(* CoDeSys 2.3.9.62 project: furrestaurantecasidefinitivo.pro *)
(* Libraries: Standard.lib 4.10.05 13:14:46, IecSfc.lib 2.6.14 11:37:46, SYSLIBCALLBACK.LIB 26.9.08 17:43:52 *)

(* Global variable list: Global_Variables *)
VAR_GLOBAL
	(*VISUALIZACION_PLATOS*)
	plato:ARRAY [1..8] OF elemento2d;
	pistonx:INT;
	vpist:INT := 3;
	velp:INT := 3;
		(*ACTUADORES CINTAS*)
		CIN_ENT_COC:BOOL;
		CIN_CLA:BOOL;
		CIN_H1:BOOL;
		CIN_H2:BOOL;
		CIN_H3:BOOL;
		CIN_SERVIR:BOOL;
		CIN_H1_A_REAL:BOOL;
		CIN_H2_A_REAL:BOOL;
		CIN_H3_A_REAL:BOOL;
		CIN_REALIM:BOOL;
		CIN_COLA_SERV:BOOL;
		(*ACTUADORES PISTON Y PROCESOS*)
		PISCLA_MAS:BOOL;
		PISCLA_MENOS:BOOL;
		AGARRAR:BOOL;
		H1:BOOL;
		H2:BOOL;
		H3:BOOL;
		DISP_PLATO:BOOL;
			(*BOTONERA CONTROL PLATOS*)
			b1:BOOL;
			b2:BOOL;
			b3:BOOL;
			b4:BOOL;
			b5:BOOL;
			b6:BOOL;
			b7:BOOL;
			b8:BOOL;
			br1:BOOL;
			br2:BOOL;
			br3:BOOL;
			blisto:BOOL;
			bup:BOOL;
			bdown:BOOL;
			bleft:BOOL;
			bright:BOOL;
			bhide:BOOL;
			vel: INT :=1 ;
		(*SENSORES CINTAS*)
		ENT_COC:BOOL;
		SEM_ENT_COC:BOOL;
		SEM_SAL_REAL:BOOL;
		S_CLA:ARRAY [1..8] OF BOOL;
		ENT_CLA:BOOL;
		ENT_H1:BOOL;
		ENT_H2:BOOL;
		ENT_H3:BOOL;
		ENT_SERVIR:BOOL;
		ESPERA_H1:BOOL;
		ESPERA_H2:BOOL;
		ESPERA_H3:BOOL;
		ENT_REAL1:BOOL;
		ENT_REAL2:BOOL;
		ENT_REAL3:BOOL;
		SEM_H2_R:BOOL;
		SEM_H2_V:BOOL;
		SEM_H2:BOOL;
		SEM_H1_R:BOOL;
		SEM_H1_V:BOOL;
		SEM_H1:BOOL;
		SAL_R:BOOL;
		ENT_TER:BOOL;
		TER_1:BOOL;
		TER_2:BOOL;
		TER_3:BOOL;
		(*SENSORES PISTON Y PROCESOS*)
		S_H1:BOOL;
		S_H2:BOOL;
		S_H3:BOOL;
		FC_PISCLA:BOOL;
		(*INFOPLATO*)

	(*VISUALIZACIÓN AGVs*)
	x1:INT:=130;
	y1:INT;
	x2:INT:=330;
	y2:INT;

		(*ACTUADORES AGVS*)
		SERVIR_PLATO1:BOOL;
		SERVIR_PLATO2:BOOL;
		CARGAR_PLATO:ARRAY [1..3] OF BOOL;

		(*SENSORES AGVs*)
		CARGADO1:BOOL;
		CARGADO2:BOOL;

		(*ACTUADORES SALÓN*)
		MARCHA1:BOOL;
		MARCHA2:BOOL;
		BIF_ARRIBA1:BOOL;
		BIF_ABAJO1:BOOL;
		BIF_ARRIBA2:BOOL;
		BIF_ABAJO2:BOOL;
		SEM_M1:BOOL;
		SEM_M2:BOOL;
		SEM_M3:BOOL;
		SEM_M4:BOOL;
		SEM_M5:BOOL;
		SEM_M6:BOOL;
		SEM_M7:BOOL;
		SEM_M8:BOOL;

		(*SENSORES SALÓN*)

		PC1_1:BOOL;
		PC1_2:BOOL;
		PR1_3:BOOL;
		PR1_2:BOOL;
		PR1_1:BOOL;
		BIF1_12:BOOL;
		BIF1_34:BOOL;
		BIF1_56:BOOL;
		BIF1_78:BOOL;

		PC2_1:BOOL;
		PC2_2:BOOL;
		PR2_3:BOOL;
		PR2_2:BOOL;
		PR2_1:BOOL;
		BIF2_12:BOOL;
		BIF2_34:BOOL;
		BIF2_56:BOOL;
		BIF2_78:BOOL;

		PS_1:BOOL;
		PS_2:BOOL;
		PS_3:BOOL;
		PS_4:BOOL;
		PS_5:BOOL;
		PS_6:BOOL;
		PS_7:BOOL;
		PS_8:BOOL;

		SS_PS_1:BOOL;
		SS_PS_2:BOOL;
		SS_PS_3:BOOL;
		SS_PS_4:BOOL;
		SS_PS_5:BOOL;
		SS_PS_6:BOOL;
		SS_PS_7:BOOL;
		SS_PS_8:BOOL;
		SS_F:BOOL;

	(*VISUALIZACION SALON*)
	ESTADO_MESA:ARRAY [1..8] OF BOOL;

		(*COLAS*)
		PENDIENTES_ENTRAR:ARRAY [1..20] OF INT;
		MESA_PEDIDO:ARRAY [1..20,1..2] OF INT;
		PEDIDO1:BOOL;
		PEDIDO2:BOOL;
		PEDIDO3:BOOL;
		MESA1:BOOL;
		MESA2:BOOL;
		MESA3:BOOL;
		MESA4:BOOL;
		MESA5:BOOL;
		MESA6:BOOL;
		MESA7:BOOL;
		MESA8:BOOL;

		(*BOTONERA COLAS*)
		B_CANCELAR:BOOL;
		B_PEDIR:BOOL;
		B_MESA:ARRAY [1..8] OF BOOL;
		B_PEDIDO:ARRAY [1..3] OF BOOL;




(*VARIABLES AUXILIARES*)
	LLENO:BOOL;
	ESPERA_ENTCOC:BOOL;
	ESPERA_CLA:BOOL;
	ESPERA_CINH1:BOOL;
	ESPERA_CINH2:BOOL;
	ESPERA_CINH3:BOOL;
	ESPERA_REAL:BOOL;
	ESPERA_SERVIR:BOOL;
	PASAH1:BOOL;
	PASAH2:BOOL;
	PASAH3:BOOL;
	H1OK:BOOL;
	H2OK:BOOL;
	H3OK:BOOL;
	SALE_REAL:BOOL;
	DIR_PISTON:ARRAY[1..8] OF INT;
	TDISP:BOOL;
	PLATO_SEM_H2:BOOL;
	PLATO_SEM_H1:BOOL;
	OC2:BOOL;
	OC1:BOOL;
	SCLAAUX:BOOL;
	REALIMENTANDO:BOOL;
	TIEMPODISP:BOOL;
END_VAR

(* Data type *)
TYPE elemento2d :
STRUCT
	x:INT;
	y:INT;
	P1:INT;
	P2:INT;
	P3:INT;
	REC:INT;
	on:BOOL;
	listo:BOOL;
	receta:STRING(5); (*temporal, solo se usara en la visualizacion*)
END_STRUCT
END_TYPE

(* POU PLC_PRG, ST *)
PROGRAM PLC_PRG
VAR
END_VAR
INFO_PLATOS;
CONTADORES;
SEMAFORO_SALIDA_H2;
SEMAFORO_SALIDA_H1;
SEMAFORO_ENTCOC;
PROCESOS;
PISTON;
CONTROL_CINTAS;
CINTA_COLA;
VIS_BOTON_PLATO;
VIS_MESAS;
VIS_PISTON;
VIS_CINTAS_PLATO;
VIS_AGV;
COLAS_PEDIDOS;
END_PROGRAM

(* POU INFO_PLATOS, ST *)
PROGRAM INFO_PLATOS
VAR
	R1:ARRAY[1..3] OF INT:=1,2,3;
	R2:ARRAY[1..3] OF INT:=2,1,3;
	R3:ARRAY[1..3] OF INT:=3,2,1;
	FS_SCLA:ARRAY[1..8] OF BOOL;
	i:INT:=1;
	i2:INT:=1;
	j:INT:=1;
	k:INT:=1;
	t:INT:=1;
	p:INT:=1;
	FLAG_DIR:BOOL;
	DISPLIBRE: BOOL:=TRUE;
	FS_DISPPLATO: BOOL;
	FB_AGARRAR:BOOL;
END_VAR
(*Asignación de receta a plato desde cola y actualización de la misma*)

IF FS_DISPPLATO=TRUE THEN
	FS_DISPPLATO:=FALSE;
	DISP_PLATO:=FALSE;
END_IF

IF NOT DISPLIBRE AND TIEMPODISP THEN
	DISPLIBRE:=TRUE;
END_IF

IF PENDIENTES_ENTRAR[1]<>0 THEN
	plato[j].REC:=PENDIENTES_ENTRAR[1];
	FOR i:=2 TO 20 BY 1 DO
		PENDIENTES_ENTRAR[i-1]:=PENDIENTES_ENTRAR[i];
	END_FOR
	PENDIENTES_ENTRAR[20]:=0;

	IF plato[j].REC=1 THEN
		plato[j].P1:=R1[1];
		plato[j].P2:=R1[2];
		plato[j].P3:=R1[3];
		plato[j].receta:='R1';
	ELSIF plato[j].REC=2 THEN
		plato[j].P1:=R2[1];
		plato[j].P2:=R2[2];
		plato[j].P3:=R2[3];
		plato[j].receta:='R2';
	ELSIF plato[j].REC=3 THEN
		plato[j].P1:=R3[1];
		plato[j].P2:=R3[2];
		plato[j].P3:=R3[3];
		plato[j].receta:='R3';
	END_IF
	IF j<8 THEN
		j:=j+1;
	ELSE
		j:=1;
	END_IF
END_IF

IF NOT LLENO AND FC_PISCLA AND NOT ENT_CLA AND DISPLIBRE AND plato[i2].P1<>0 THEN
	DISP_PLATO:=TRUE;
	FS_DISPPLATO:=TRUE;
	DISPLIBRE:=FALSE;
	IF i2<8 THEN
		i2:=i2+1;
	ELSE
		i2:=1;
	END_IF
END_IF



(*Manejo del sensor de clasificación S_CLA y comunicación con el pistón*)

FOR t:=1 TO 8 BY 1 DO
	IF S_CLA[t]=TRUE AND FS_SCLA[t]=FALSE THEN
		FS_SCLA[t]:=TRUE;
		IF plato[t].P1<>0 THEN
			FOR k:=1 TO 8 BY 1 DO
				IF DIR_PISTON[k]=0 AND FLAG_DIR=FALSE THEN
					DIR_PISTON[k]:=plato[t].P1;
					FLAG_DIR:=TRUE;
				END_IF
			END_FOR
			FLAG_DIR:=FALSE;
			plato[t].P1:=0;
		ELSIF plato[t].P1=0 AND plato[t].P2<>0 THEN
			FOR k:=1 TO 8 BY 1 DO
				IF DIR_PISTON[k]=0 AND FLAG_DIR=FALSE THEN
					DIR_PISTON[k]:=plato[t].P2;
					FLAG_DIR:=TRUE;
				END_IF
			END_FOR
			FLAG_DIR:=FALSE;
			plato[t].P2:=0;
		ELSIF plato[t].P1=0 AND plato[t].P2=0 AND plato[t].P3<>0 THEN
			FOR k:=1 TO 8 BY 1 DO
				IF DIR_PISTON[k]=0 AND FLAG_DIR=FALSE THEN
					DIR_PISTON[k]:=plato[t].P3;
					FLAG_DIR:=TRUE;
				END_IF
			END_FOR
			FLAG_DIR:=FALSE;
			plato[t].P3:=0;
		ELSIF plato[t].P1=0 AND plato[t].P2=0 AND plato[t].P3=0 AND plato[t].REC<>0 THEN
			FOR k:=1 TO 8 BY 1 DO
				IF DIR_PISTON[k]=0 AND FLAG_DIR=FALSE THEN
					DIR_PISTON[k]:=4;
					FLAG_DIR:=TRUE;
					plato[t].listo:=TRUE;
				END_IF
			END_FOR
			FLAG_DIR:=FALSE;
			plato[t].REC:=0;
		END_IF
	ELSIF S_CLA[t]=FALSE THEN
		FS_SCLA[t]:=FALSE;
	END_IF
END_FOR

(*Manejo de la cola del pistón*)




IF NOT AGARRAR AND NOT FB_AGARRAR THEN
	FOR p:=2 TO 8 BY 1 DO
		DIR_PISTON[p-1]:=DIR_PISTON[p];
	END_FOR
	DIR_PISTON[8]:=0;
	FB_AGARRAR:=TRUE;
ELSIF AGARRAR THEN
	FB_AGARRAR:=FALSE;
END_IF
END_PROGRAM

(* POU CONTADORES, LD *)
PROGRAM CONTADORES
VAR
	NUM_ENTCOC: CTUD;
	NUM_COCINA: CTUD;
	NUM_CLA: CTUD;
	FB_ENTCOC1: F_TRIG;
	FB_ENTCOC2: F_TRIG;
	NUM_H1: CTUD;
	NUM_H2: CTUD;
	NUM_H3: CTUD;
	NUM_REAL: CTUD;
	RET_SALREAL: TOF;
	FS_ENTH3: R_TRIG;
	FS_ENTH2: R_TRIG;
	FS_ENTH1: R_TRIG;
	FS_SALEREAL: R_TRIG;
	FS_ENTSERVIR: R_TRIG;
	NUM_SERVIR: CTUD;
	SEPARACION_PLATOS_DISP: TOF;
	ENTRA_SMF_H2: R_TRIG;
	NUM_SMF_H2: CTUD;
	ENTRA_SMF_H1: R_TRIG;
	NUM_SMF_H1: CTUD;
	TSEMAFORO2: TON;
	TSEMAFORO1: TON;
	FS_ENTREAL1: R_TRIG;
	FS_ENTREAL2: R_TRIG;
	FS_ENTREAL3: R_TRIG;
	FB_SALR: F_TRIG;
	FB_DISPPLATO: F_TRIG;
	tiempo_disp: TON;
END_VAR
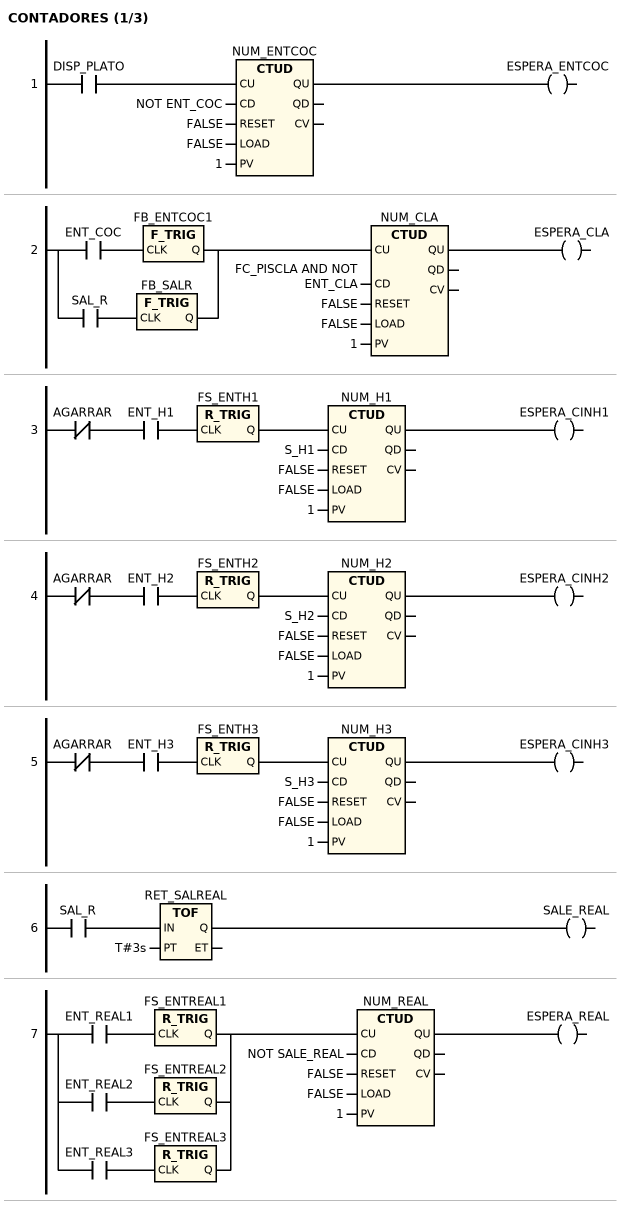
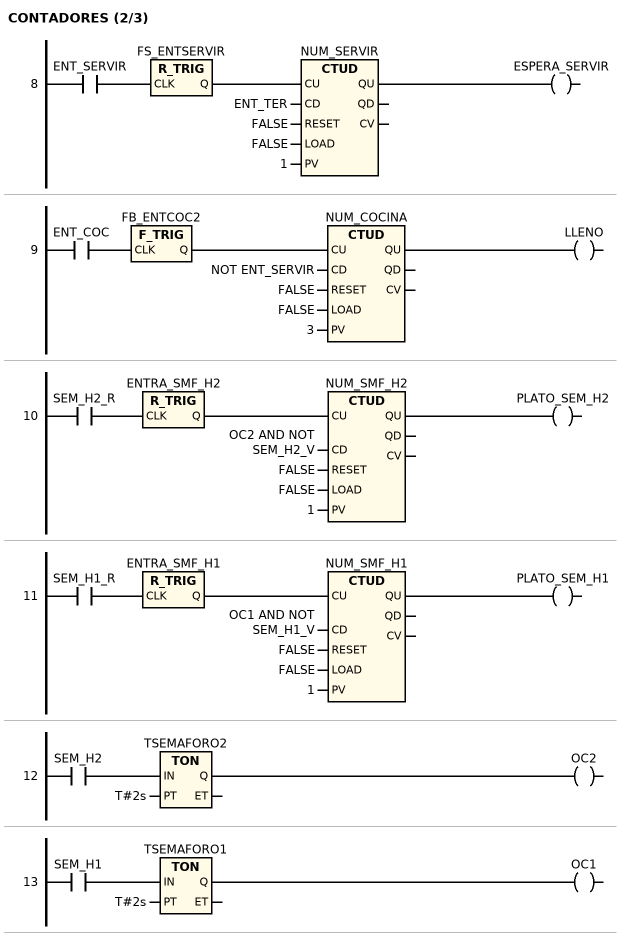
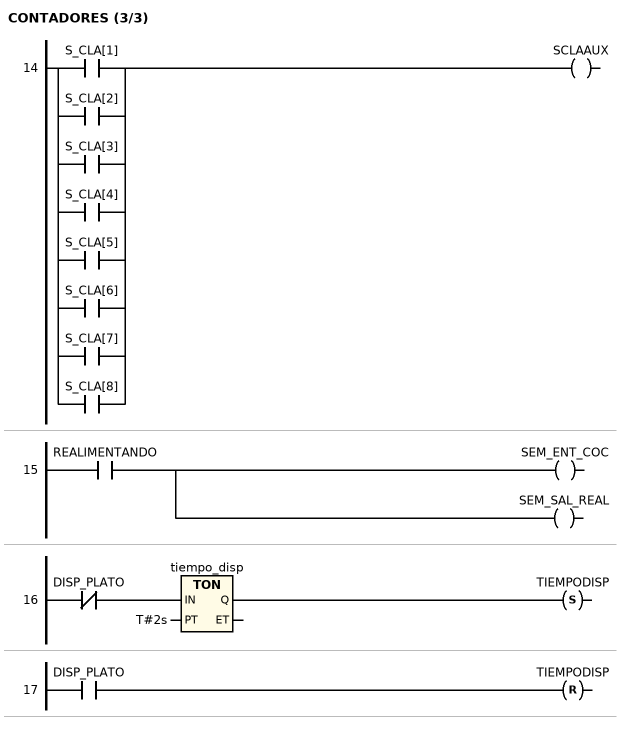
_LD_ (* Ladder Diagram *)
NETWORK 1
	[DISP_PLATO] - NUM_ENTCOC:CTUD(CU: *, CD: NOT ENT_COC, RESET: FALSE, LOAD: FALSE, PV: 1) --- (ESPERA_ENTCOC)
NETWORK 2
	{ [ENT_COC] - FB_ENTCOC1:F_TRIG(CLK: *) | [SAL_R] - FB_SALR:F_TRIG(CLK: *) } - NUM_CLA:CTUD(CU: *, CD: FC_PISCLA AND NOT ENT_CLA, RESET: FALSE, LOAD: FALSE, PV: 1) --- (ESPERA_CLA)
NETWORK 3
	[/AGARRAR] - [ENT_H1] - FS_ENTH1:R_TRIG(CLK: *) - NUM_H1:CTUD(CU: *, CD: S_H1, RESET: FALSE, LOAD: FALSE, PV: 1) --- (ESPERA_CINH1)
NETWORK 4
	[/AGARRAR] - [ENT_H2] - FS_ENTH2:R_TRIG(CLK: *) - NUM_H2:CTUD(CU: *, CD: S_H2, RESET: FALSE, LOAD: FALSE, PV: 1) --- (ESPERA_CINH2)
NETWORK 5
	[/AGARRAR] - [ENT_H3] - FS_ENTH3:R_TRIG(CLK: *) - NUM_H3:CTUD(CU: *, CD: S_H3, RESET: FALSE, LOAD: FALSE, PV: 1) --- (ESPERA_CINH3)
NETWORK 6
	[SAL_R] - RET_SALREAL:TOF(IN: *, PT: T#3s) --- (SALE_REAL)
NETWORK 7
	{ [ENT_REAL1] - FS_ENTREAL1:R_TRIG(CLK: *) | [ENT_REAL2] - FS_ENTREAL2:R_TRIG(CLK: *) | [ENT_REAL3] - FS_ENTREAL3:R_TRIG(CLK: *) } - NUM_REAL:CTUD(CU: *, CD: NOT SALE_REAL, RESET: FALSE, LOAD: FALSE, PV: 1) --- (ESPERA_REAL)
NETWORK 8
	[ENT_SERVIR] - FS_ENTSERVIR:R_TRIG(CLK: *) - NUM_SERVIR:CTUD(CU: *, CD: ENT_TER, RESET: FALSE, LOAD: FALSE, PV: 1) --- (ESPERA_SERVIR)
NETWORK 9
	[ENT_COC] - FB_ENTCOC2:F_TRIG(CLK: *) - NUM_COCINA:CTUD(CU: *, CD: NOT ENT_SERVIR, RESET: FALSE, LOAD: FALSE, PV: 3) --- (LLENO)
NETWORK 10
	[SEM_H2_R] - ENTRA_SMF_H2:R_TRIG(CLK: *) - NUM_SMF_H2:CTUD(CU: *, CD: OC2 AND NOT SEM_H2_V, RESET: FALSE, LOAD: FALSE, PV: 1) --- (PLATO_SEM_H2)
NETWORK 11
	[SEM_H1_R] - ENTRA_SMF_H1:R_TRIG(CLK: *) - NUM_SMF_H1:CTUD(CU: *, CD: OC1 AND NOT SEM_H1_V, RESET: FALSE, LOAD: FALSE, PV: 1) --- (PLATO_SEM_H1)
NETWORK 12
	[SEM_H2] - TSEMAFORO2:TON(IN: *, PT: T#2s) --- (OC2)
NETWORK 13
	[SEM_H1] - TSEMAFORO1:TON(IN: *, PT: T#2s) --- (OC1)
NETWORK 14
	{ [S_CLA[1]] | [S_CLA[2]] | [S_CLA[3]] | [S_CLA[4]] | [S_CLA[5]] | [S_CLA[6]] | [S_CLA[7]] | [S_CLA[8]] } --- (SCLAAUX)
NETWORK 15
	[REALIMENTANDO] --- (SEM_ENT_COC) (SEM_SAL_REAL)
NETWORK 16
	[/DISP_PLATO] - tiempo_disp:TON(IN: *, PT: T#2s) --- (S TIEMPODISP)
NETWORK 17
	[DISP_PLATO] --- (R TIEMPODISP)
_END_LD_
(* the same logic as Structured Text *)
(* Network 1 *)
NUM_ENTCOC(CU := DISP_PLATO, CD := NOT ENT_COC, RESET := FALSE, LOAD := FALSE, PV := 1);
ESPERA_ENTCOC := NUM_ENTCOC.QU;
(* Network 2 *)
FB_ENTCOC1(CLK := ENT_COC);
FB_SALR(CLK := SAL_R);
NUM_CLA(CU := FB_ENTCOC1.Q OR FB_SALR.Q, CD := FC_PISCLA AND NOT ENT_CLA, RESET := FALSE, LOAD := FALSE, PV := 1);
ESPERA_CLA := NUM_CLA.QU;
(* Network 3 *)
FS_ENTH1(CLK := NOT AGARRAR AND ENT_H1);
NUM_H1(CU := FS_ENTH1.Q, CD := S_H1, RESET := FALSE, LOAD := FALSE, PV := 1);
ESPERA_CINH1 := NUM_H1.QU;
(* Network 4 *)
FS_ENTH2(CLK := NOT AGARRAR AND ENT_H2);
NUM_H2(CU := FS_ENTH2.Q, CD := S_H2, RESET := FALSE, LOAD := FALSE, PV := 1);
ESPERA_CINH2 := NUM_H2.QU;
(* Network 5 *)
FS_ENTH3(CLK := NOT AGARRAR AND ENT_H3);
NUM_H3(CU := FS_ENTH3.Q, CD := S_H3, RESET := FALSE, LOAD := FALSE, PV := 1);
ESPERA_CINH3 := NUM_H3.QU;
(* Network 6 *)
RET_SALREAL(IN := SAL_R, PT := T#3s);
SALE_REAL := RET_SALREAL.Q;
(* Network 7 *)
FS_ENTREAL1(CLK := ENT_REAL1);
FS_ENTREAL2(CLK := ENT_REAL2);
FS_ENTREAL3(CLK := ENT_REAL3);
NUM_REAL(CU := FS_ENTREAL1.Q OR FS_ENTREAL2.Q OR FS_ENTREAL3.Q, CD := NOT SALE_REAL, RESET := FALSE, LOAD := FALSE, PV := 1);
ESPERA_REAL := NUM_REAL.QU;
(* Network 8 *)
FS_ENTSERVIR(CLK := ENT_SERVIR);
NUM_SERVIR(CU := FS_ENTSERVIR.Q, CD := ENT_TER, RESET := FALSE, LOAD := FALSE, PV := 1);
ESPERA_SERVIR := NUM_SERVIR.QU;
(* Network 9 *)
FB_ENTCOC2(CLK := ENT_COC);
NUM_COCINA(CU := FB_ENTCOC2.Q, CD := NOT ENT_SERVIR, RESET := FALSE, LOAD := FALSE, PV := 3);
LLENO := NUM_COCINA.QU;
(* Network 10 *)
ENTRA_SMF_H2(CLK := SEM_H2_R);
NUM_SMF_H2(CU := ENTRA_SMF_H2.Q, CD := OC2 AND NOT SEM_H2_V, RESET := FALSE, LOAD := FALSE, PV := 1);
PLATO_SEM_H2 := NUM_SMF_H2.QU;
(* Network 11 *)
ENTRA_SMF_H1(CLK := SEM_H1_R);
NUM_SMF_H1(CU := ENTRA_SMF_H1.Q, CD := OC1 AND NOT SEM_H1_V, RESET := FALSE, LOAD := FALSE, PV := 1);
PLATO_SEM_H1 := NUM_SMF_H1.QU;
(* Network 12 *)
TSEMAFORO2(IN := SEM_H2, PT := T#2s);
OC2 := TSEMAFORO2.Q;
(* Network 13 *)
TSEMAFORO1(IN := SEM_H1, PT := T#2s);
OC1 := TSEMAFORO1.Q;
(* Network 14 *)
SCLAAUX := S_CLA[1] OR S_CLA[2] OR S_CLA[3] OR S_CLA[4] OR S_CLA[5] OR S_CLA[6] OR S_CLA[7] OR S_CLA[8];
(* Network 15 *)
SEM_ENT_COC := REALIMENTANDO;
SEM_SAL_REAL := REALIMENTANDO;
(* Network 16 *)
tiempo_disp(IN := NOT DISP_PLATO, PT := T#2s);
IF tiempo_disp.Q THEN TIEMPODISP := TRUE; END_IF;
(* Network 17 *)
IF DISP_PLATO THEN TIEMPODISP := FALSE; END_IF;
END_PROGRAM

(* POU SEMAFORO_SALIDA_H2, SFC *)
PROGRAM SEMAFORO_SALIDA_H2
VAR
END_VAR
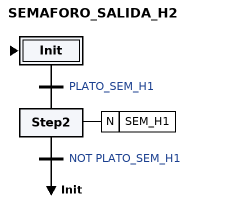
INITIAL_STEP Init:
END_STEP
TRANSITION FROM Init TO Step2 := PLATO_SEM_H1;
END_TRANSITION
STEP Step2:
	SEM_H1(N);
END_STEP
TRANSITION FROM Step2 TO Init := NOT PLATO_SEM_H1;
END_TRANSITION
END_PROGRAM

(* POU SEMAFORO_SALIDA_H1, SFC *)
PROGRAM SEMAFORO_SALIDA_H1
VAR
END_VAR
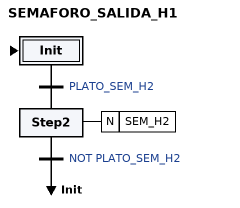
INITIAL_STEP Init:
END_STEP
TRANSITION FROM Init TO Step2 := PLATO_SEM_H2;
END_TRANSITION
STEP Step2:
	SEM_H2(N);
END_STEP
TRANSITION FROM Step2 TO Init := NOT PLATO_SEM_H2;
END_TRANSITION
END_PROGRAM

(* POU SEMAFORO_ENTCOC, SFC *)
PROGRAM SEMAFORO_ENTCOC
VAR
	FB_SALR: F_TRIG;
	FB_SCLAAUX: F_TRIG;
END_VAR
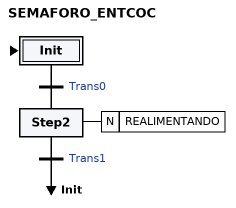
INITIAL_STEP Init:
END_STEP
TRANSITION FROM Init TO Step2 := Trans0;
END_TRANSITION
STEP Step2:
	REALIMENTANDO(N);
END_STEP
TRANSITION FROM Step2 TO Init := Trans1;
END_TRANSITION

TRANSITION Trans0:
_LD_ (* Ladder Diagram *)
NETWORK 1
	[SAL_R] - FB_SALR:F_TRIG(CLK: *)
_END_LD_
(* the same logic as Structured Text *)
(* Network 1 *)
FB_SALR(CLK := SAL_R);
Trans0 := FB_SALR.Q;
END_TRANSITION

TRANSITION Trans1:
_LD_ (* Ladder Diagram *)
NETWORK 1
	[SCLAAUX] - FB_SCLAAUX:F_TRIG(CLK: *)
_END_LD_
(* the same logic as Structured Text *)
(* Network 1 *)
FB_SCLAAUX(CLK := SCLAAUX);
Trans1 := FB_SCLAAUX.Q;
END_TRANSITION
END_PROGRAM

(* POU PROCESOS, LD *)
PROGRAM PROCESOS
VAR
	PROCESO_H1: FB_PROCESOS;
	PROCESO_H2: FB_PROCESOS;
	PROCESO_H3: FB_PROCESOS;
END_VAR
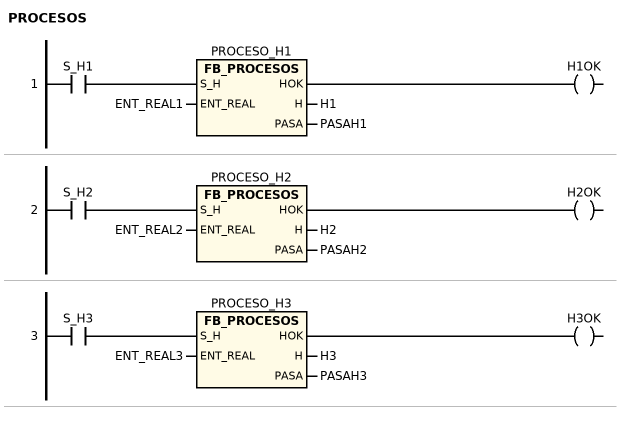
_LD_ (* Ladder Diagram *)
NETWORK 1
	[S_H1] - PROCESO_H1:FB_PROCESOS(S_H: *, ENT_REAL: ENT_REAL1, H => H1, PASA => PASAH1) --- (H1OK)
NETWORK 2
	[S_H2] - PROCESO_H2:FB_PROCESOS(S_H: *, ENT_REAL: ENT_REAL2, H => H2, PASA => PASAH2) --- (H2OK)
NETWORK 3
	[S_H3] - PROCESO_H3:FB_PROCESOS(S_H: *, ENT_REAL: ENT_REAL3, H => H3, PASA => PASAH3) --- (H3OK)
_END_LD_
(* the same logic as Structured Text *)
(* Network 1 *)
PROCESO_H1(S_H := S_H1, ENT_REAL := ENT_REAL1);
H1 := PROCESO_H1.H;
PASAH1 := PROCESO_H1.PASA;
H1OK := PROCESO_H1.HOK;
(* Network 2 *)
PROCESO_H2(S_H := S_H2, ENT_REAL := ENT_REAL2);
H2 := PROCESO_H2.H;
PASAH2 := PROCESO_H2.PASA;
H2OK := PROCESO_H2.HOK;
(* Network 3 *)
PROCESO_H3(S_H := S_H3, ENT_REAL := ENT_REAL3);
H3 := PROCESO_H3.H;
PASAH3 := PROCESO_H3.PASA;
H3OK := PROCESO_H3.HOK;
END_PROGRAM

(* POU FB_PROCESOS, SFC *)
FUNCTION_BLOCK FB_PROCESOS
VAR_INPUT
	S_H:BOOL;
	ENT_REAL:BOOL;
END_VAR
VAR_OUTPUT
	HOK:BOOL;
	H:BOOL;
	PASA:BOOL;
END_VAR
VAR
	ESPERA_PROCESO: TON;
END_VAR
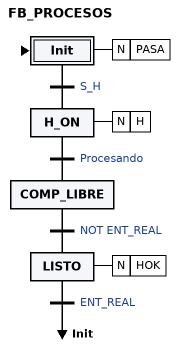
INITIAL_STEP Init:
	PASA(N);
END_STEP
TRANSITION FROM Init TO H_ON := S_H;
END_TRANSITION
STEP H_ON:
	H(N);
END_STEP
TRANSITION FROM H_ON TO COMP_LIBRE  := Procesando;
END_TRANSITION
STEP COMP_LIBRE :
END_STEP
TRANSITION FROM COMP_LIBRE  TO LISTO := NOT ENT_REAL;
END_TRANSITION
STEP LISTO:
	HOK(N);
END_STEP
TRANSITION FROM LISTO TO Init := ENT_REAL;
END_TRANSITION

TRANSITION Procesando:
_LD_ (* Ladder Diagram *)
NETWORK 1
	[H] - ESPERA_PROCESO:TON(IN: *, PT: T#5s)
_END_LD_
(* the same logic as Structured Text *)
(* Network 1 *)
ESPERA_PROCESO(IN := H, PT := T#5s);
Procesando := ESPERA_PROCESO.Q;
END_TRANSITION
END_FUNCTION_BLOCK

(* POU PISTON, SFC *)
PROGRAM PISTON
VAR
END_VAR
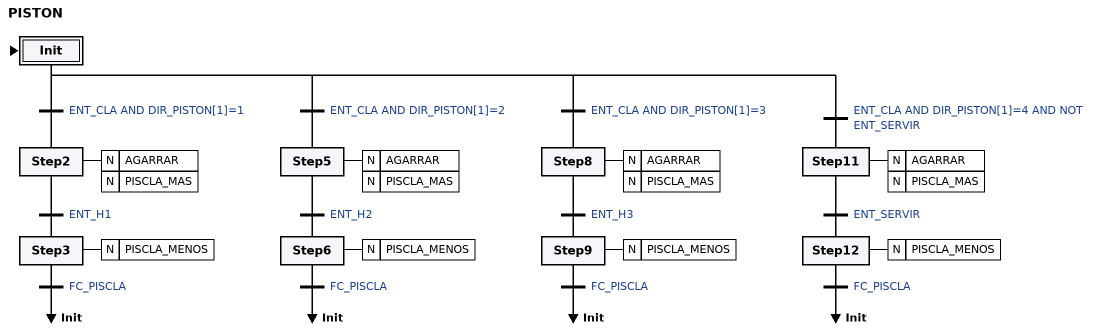
INITIAL_STEP Init:
END_STEP
TRANSITION FROM Init TO Step2 := ENT_CLA AND DIR_PISTON[1]=1;
END_TRANSITION
TRANSITION FROM Init TO Step5 := ENT_CLA AND DIR_PISTON[1]=2;
END_TRANSITION
TRANSITION FROM Init TO Step8 := ENT_CLA AND DIR_PISTON[1]=3;
END_TRANSITION
TRANSITION FROM Init TO Step11 := ENT_CLA AND DIR_PISTON[1]=4 AND NOT ENT_SERVIR;
END_TRANSITION
STEP Step2:
	AGARRAR(N);
	PISCLA_MAS(N);
END_STEP
TRANSITION FROM Step2 TO Step3 := ENT_H1;
END_TRANSITION
STEP Step3:
	PISCLA_MENOS(N);
END_STEP
TRANSITION FROM Step3 TO Init := FC_PISCLA;
END_TRANSITION
STEP Step5:
	AGARRAR(N);
	PISCLA_MAS(N);
END_STEP
TRANSITION FROM Step5 TO Step6 := ENT_H2;
END_TRANSITION
STEP Step6:
	PISCLA_MENOS(N);
END_STEP
TRANSITION FROM Step6 TO Init := FC_PISCLA;
END_TRANSITION
STEP Step8:
	AGARRAR(N);
	PISCLA_MAS(N);
END_STEP
TRANSITION FROM Step8 TO Step9 := ENT_H3;
END_TRANSITION
STEP Step9:
	PISCLA_MENOS(N);
END_STEP
TRANSITION FROM Step9 TO Init := FC_PISCLA;
END_TRANSITION
STEP Step11:
	AGARRAR(N);
	PISCLA_MAS(N);
END_STEP
TRANSITION FROM Step11 TO Step12 := ENT_SERVIR;
END_TRANSITION
STEP Step12:
	PISCLA_MENOS(N);
END_STEP
TRANSITION FROM Step12 TO Init := FC_PISCLA;
END_TRANSITION
END_PROGRAM

(* POU CONTROL_CINTAS, LD *)
PROGRAM CONTROL_CINTAS
VAR
	CINTA_H1_A_REAL: FB_CINTAS_H_A_REAL;
	CINTA_H2_A_REAL: FB_CINTAS_H_A_REAL;
	CINTA_H3_A_REAL: FB_CINTAS_H_A_REAL;
	FS_TER3: R_TRIG;
	FS_TER2: R_TRIG;
	FS_TER1: R_TRIG;
	FS_TER1_1: R_TRIG;
	FS_TER2_1: R_TRIG;
	FS_TER3_1: R_TRIG;
END_VAR
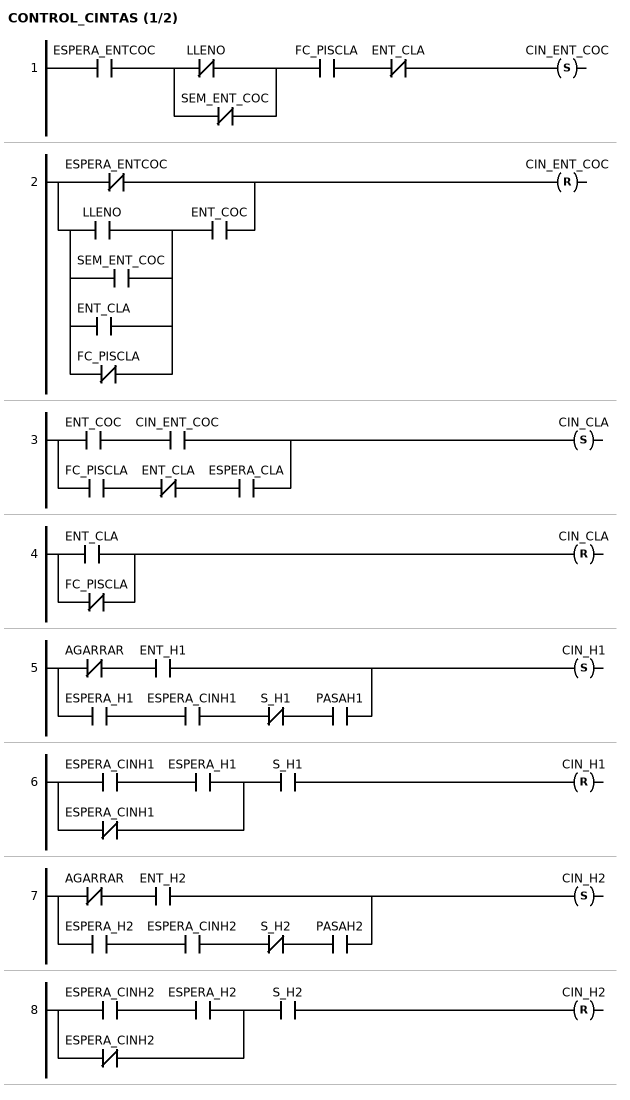
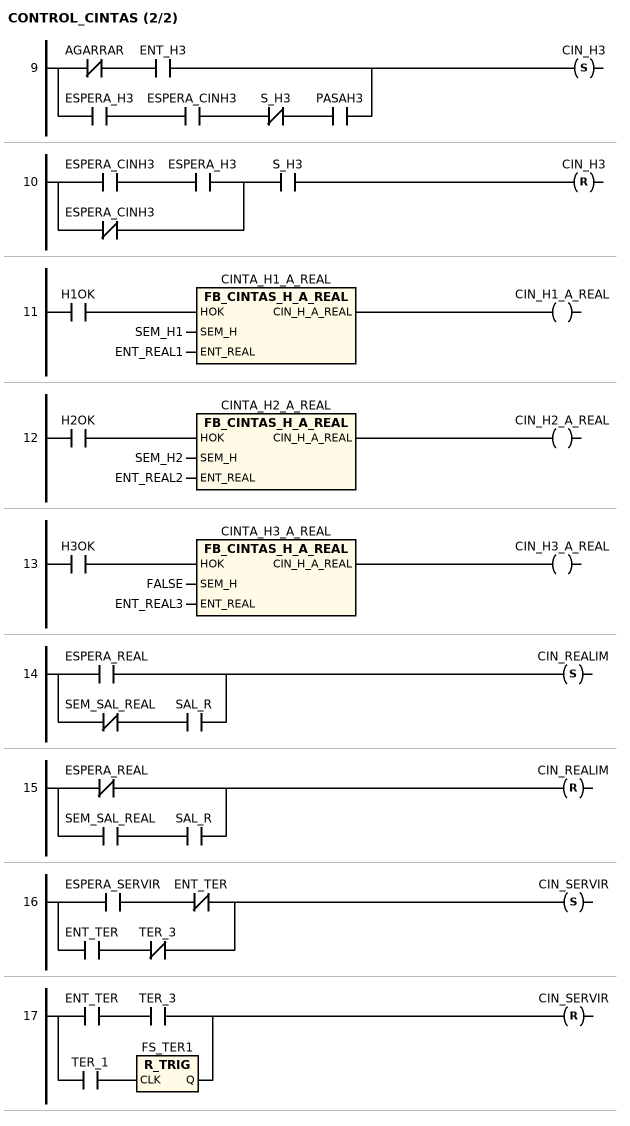
_LD_ (* Ladder Diagram *)
NETWORK 1
	[ESPERA_ENTCOC] - { [/LLENO] | [/SEM_ENT_COC] } - [FC_PISCLA] - [/ENT_CLA] --- (S CIN_ENT_COC)
NETWORK 2
	{ [/ESPERA_ENTCOC] | { [LLENO] | [SEM_ENT_COC] | [ENT_CLA] | [/FC_PISCLA] } - [ENT_COC] } --- (R CIN_ENT_COC)
NETWORK 3
	{ [ENT_COC] - [CIN_ENT_COC] | [FC_PISCLA] - [/ENT_CLA] - [ESPERA_CLA] } --- (S CIN_CLA)
NETWORK 4
	{ [ENT_CLA] | [/FC_PISCLA] } --- (R CIN_CLA)
NETWORK 5
	{ [/AGARRAR] - [ENT_H1] | [ESPERA_H1] - [ESPERA_CINH1] - [/S_H1] - [PASAH1] } --- (S CIN_H1)
NETWORK 6
	{ [ESPERA_CINH1] - [ESPERA_H1] | [/ESPERA_CINH1] } - [S_H1] --- (R CIN_H1)
NETWORK 7
	{ [/AGARRAR] - [ENT_H2] | [ESPERA_H2] - [ESPERA_CINH2] - [/S_H2] - [PASAH2] } --- (S CIN_H2)
NETWORK 8
	{ [ESPERA_CINH2] - [ESPERA_H2] | [/ESPERA_CINH2] } - [S_H2] --- (R CIN_H2)
NETWORK 9
	{ [/AGARRAR] - [ENT_H3] | [ESPERA_H3] - [ESPERA_CINH3] - [/S_H3] - [PASAH3] } --- (S CIN_H3)
NETWORK 10
	{ [ESPERA_CINH3] - [ESPERA_H3] | [/ESPERA_CINH3] } - [S_H3] --- (R CIN_H3)
NETWORK 11
	[H1OK] - CINTA_H1_A_REAL:FB_CINTAS_H_A_REAL(HOK: *, SEM_H: SEM_H1, ENT_REAL: ENT_REAL1) --- (CIN_H1_A_REAL)
NETWORK 12
	[H2OK] - CINTA_H2_A_REAL:FB_CINTAS_H_A_REAL(HOK: *, SEM_H: SEM_H2, ENT_REAL: ENT_REAL2) --- (CIN_H2_A_REAL)
NETWORK 13
	[H3OK] - CINTA_H3_A_REAL:FB_CINTAS_H_A_REAL(HOK: *, SEM_H: FALSE, ENT_REAL: ENT_REAL3) --- (CIN_H3_A_REAL)
NETWORK 14
	{ [ESPERA_REAL] | [/SEM_SAL_REAL] - [SAL_R] } --- (S CIN_REALIM)
NETWORK 15
	{ [/ESPERA_REAL] | [SEM_SAL_REAL] - [SAL_R] } --- (R CIN_REALIM)
NETWORK 16
	{ [ESPERA_SERVIR] - [/ENT_TER] | [ENT_TER] - [/TER_3] } --- (S CIN_SERVIR)
NETWORK 17
	{ [ENT_TER] - [TER_3] | [TER_1] - FS_TER1:R_TRIG(CLK: *) } --- (R CIN_SERVIR)
_END_LD_
(* the same logic as Structured Text *)
(* Network 1 *)
IF ESPERA_ENTCOC AND (NOT LLENO OR NOT SEM_ENT_COC) AND FC_PISCLA AND NOT ENT_CLA THEN CIN_ENT_COC := TRUE; END_IF;
(* Network 2 *)
IF NOT ESPERA_ENTCOC OR (LLENO OR SEM_ENT_COC OR ENT_CLA OR NOT FC_PISCLA) AND ENT_COC THEN CIN_ENT_COC := FALSE; END_IF;
(* Network 3 *)
IF ENT_COC AND CIN_ENT_COC OR FC_PISCLA AND NOT ENT_CLA AND ESPERA_CLA THEN CIN_CLA := TRUE; END_IF;
(* Network 4 *)
IF ENT_CLA OR NOT FC_PISCLA THEN CIN_CLA := FALSE; END_IF;
(* Network 5 *)
IF NOT AGARRAR AND ENT_H1 OR ESPERA_H1 AND ESPERA_CINH1 AND NOT S_H1 AND PASAH1 THEN CIN_H1 := TRUE; END_IF;
(* Network 6 *)
IF (ESPERA_CINH1 AND ESPERA_H1 OR NOT ESPERA_CINH1) AND S_H1 THEN CIN_H1 := FALSE; END_IF;
(* Network 7 *)
IF NOT AGARRAR AND ENT_H2 OR ESPERA_H2 AND ESPERA_CINH2 AND NOT S_H2 AND PASAH2 THEN CIN_H2 := TRUE; END_IF;
(* Network 8 *)
IF (ESPERA_CINH2 AND ESPERA_H2 OR NOT ESPERA_CINH2) AND S_H2 THEN CIN_H2 := FALSE; END_IF;
(* Network 9 *)
IF NOT AGARRAR AND ENT_H3 OR ESPERA_H3 AND ESPERA_CINH3 AND NOT S_H3 AND PASAH3 THEN CIN_H3 := TRUE; END_IF;
(* Network 10 *)
IF (ESPERA_CINH3 AND ESPERA_H3 OR NOT ESPERA_CINH3) AND S_H3 THEN CIN_H3 := FALSE; END_IF;
(* Network 11 *)
CINTA_H1_A_REAL(HOK := H1OK, SEM_H := SEM_H1, ENT_REAL := ENT_REAL1);
CIN_H1_A_REAL := CINTA_H1_A_REAL.CIN_H_A_REAL;
(* Network 12 *)
CINTA_H2_A_REAL(HOK := H2OK, SEM_H := SEM_H2, ENT_REAL := ENT_REAL2);
CIN_H2_A_REAL := CINTA_H2_A_REAL.CIN_H_A_REAL;
(* Network 13 *)
CINTA_H3_A_REAL(HOK := H3OK, SEM_H := FALSE, ENT_REAL := ENT_REAL3);
CIN_H3_A_REAL := CINTA_H3_A_REAL.CIN_H_A_REAL;
(* Network 14 *)
IF ESPERA_REAL OR NOT SEM_SAL_REAL AND SAL_R THEN CIN_REALIM := TRUE; END_IF;
(* Network 15 *)
IF NOT ESPERA_REAL OR SEM_SAL_REAL AND SAL_R THEN CIN_REALIM := FALSE; END_IF;
(* Network 16 *)
IF ESPERA_SERVIR AND NOT ENT_TER OR ENT_TER AND NOT TER_3 THEN CIN_SERVIR := TRUE; END_IF;
(* Network 17 *)
FS_TER1(CLK := TER_1);
IF ENT_TER AND TER_3 OR FS_TER1.Q THEN CIN_SERVIR := FALSE; END_IF;
END_PROGRAM

(* POU FB_CINTAS_H_A_REAL, LD *)
FUNCTION_BLOCK FB_CINTAS_H_A_REAL
VAR_INPUT
	HOK:BOOL;
	SEM_H:BOOL;
	ENT_REAL:BOOL;
END_VAR
VAR_OUTPUT
	CIN_H_A_REAL:BOOL;
END_VAR
VAR
	FB_ENTREAL: F_TRIG;
END_VAR
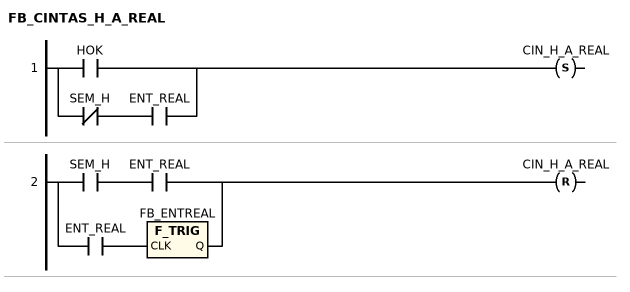
_LD_ (* Ladder Diagram *)
NETWORK 1
	{ [HOK] | [/SEM_H] - [ENT_REAL] } --- (S CIN_H_A_REAL)
NETWORK 2
	{ [SEM_H] - [ENT_REAL] | [ENT_REAL] - FB_ENTREAL:F_TRIG(CLK: *) } --- (R CIN_H_A_REAL)
_END_LD_
(* the same logic as Structured Text *)
(* Network 1 *)
IF HOK OR NOT SEM_H AND ENT_REAL THEN CIN_H_A_REAL := TRUE; END_IF;
(* Network 2 *)
FB_ENTREAL(CLK := ENT_REAL);
IF SEM_H AND ENT_REAL OR FB_ENTREAL.Q THEN CIN_H_A_REAL := FALSE; END_IF;
END_FUNCTION_BLOCK

(* POU CINTA_COLA, SFC *)
PROGRAM CINTA_COLA
VAR
END_VAR
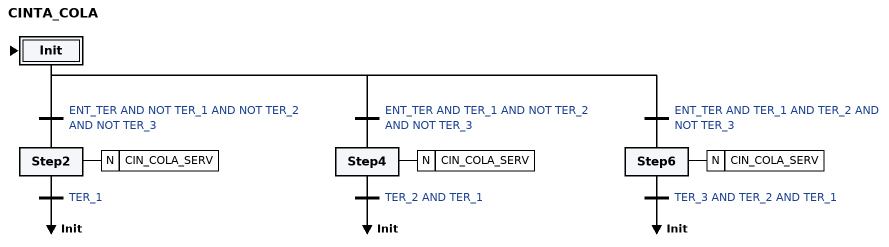
INITIAL_STEP Init:
END_STEP
TRANSITION FROM Init TO Step2 := ENT_TER AND NOT TER_1 AND NOT TER_2 AND NOT TER_3;
END_TRANSITION
TRANSITION FROM Init TO Step4 := ENT_TER AND TER_1 AND NOT TER_2 AND NOT TER_3;
END_TRANSITION
TRANSITION FROM Init TO Step6 := ENT_TER AND TER_1 AND TER_2 AND NOT TER_3;
END_TRANSITION
STEP Step2:
	CIN_COLA_SERV(N);
END_STEP
TRANSITION FROM Step2 TO Init := TER_1;
END_TRANSITION
STEP Step4:
	CIN_COLA_SERV(N);
END_STEP
TRANSITION FROM Step4 TO Init := TER_2 AND TER_1;
END_TRANSITION
STEP Step6:
	CIN_COLA_SERV(N);
END_STEP
TRANSITION FROM Step6 TO Init := TER_3 AND TER_2 AND TER_1;
END_TRANSITION
END_PROGRAM

(* POU VIS_BOTON_PLATO, ST *)
PROGRAM VIS_BOTON_PLATO
VAR
	fs_bhide:BOOL := FALSE;
	i:INT;
END_VAR
(*Botonera de movimiento manual*)
IF b1 THEN
	i:=1;
ELSIF b2 THEN
	i:=2;
ELSIF b3 THEN
	i:=3;
ELSIF b4 THEN
	i:=4;
ELSIF b5 THEN
	i:=5;
ELSIF b6 THEN
	i:=6;
ELSIF b7 THEN
	i:=7;
ELSIF b8 THEN
	i:=8;
ELSE
	i:=0;
END_IF;

IF i<>0 THEN

IF bup THEN
	plato[i].y:=plato[i].y-vel;
END_IF;

IF bdown THEN
	plato[i].y:=plato[i].y+vel;
END_IF;

IF bright THEN
	plato[i].x:=plato[i].x+vel;
END_IF;

IF bleft THEN
	plato[i].x:=plato[i].x-vel;
END_IF;

IF br1 THEN
	plato[i].receta:='R1';
END_IF;

IF br2 THEN
	plato[i].receta:='R2';
END_IF;

IF br3 THEN
	plato[i].receta:='R3';
END_IF;

IF blisto THEN
	plato[i].listo:=TRUE;
END_IF;

IF bhide THEN (*detetor de flanco de bhide*)
	IF NOT fs_bhide THEN
		plato[i].x:=0;
		plato[i].y:=0;
		plato[i].listo:=FALSE;
		plato[i].receta:='--';
		IF plato[i].on THEN
			plato[i].on:=FALSE;
		ELSE
			plato[i].on:=TRUE;
		END_IF
		fs_bhide:=TRUE;
	END_IF;
ELSE
	fs_bhide:=FALSE;
END_IF;

END_IF;
END_PROGRAM

(* POU VIS_MESAS, ST *)
PROGRAM VIS_MESAS
VAR
	i:INT;
END_VAR
FOR i:=1 TO 8 BY 1 DO
	IF B_PEDIR AND B_MESA[i] THEN
		ESTADO_MESA[i]:=TRUE;
	END_IF;
END_FOR;


IF (SERVIR_PLATO1 OR SERVIR_PLATO2) AND PS_1 THEN
	ESTADO_MESA[1]:=FALSE;
	IF SERVIR_PLATO1 THEN
		CARGADO1:=FALSE;
	ELSE
		CARGADO2:=FALSE;
	END_IF;
END_IF;

IF (SERVIR_PLATO1 OR SERVIR_PLATO2) AND PS_2 THEN
	ESTADO_MESA[2]:=FALSE;
	IF SERVIR_PLATO1 THEN
		CARGADO1:=FALSE;
	ELSE
		CARGADO2:=FALSE;
	END_IF;
END_IF;

IF (SERVIR_PLATO1 OR SERVIR_PLATO2) AND PS_3 THEN
	ESTADO_MESA[3]:=FALSE;
	IF SERVIR_PLATO1 THEN
		CARGADO1:=FALSE;
	ELSE
		CARGADO2:=FALSE;
	END_IF;
END_IF;

IF (SERVIR_PLATO1 OR SERVIR_PLATO2) AND PS_4 THEN
	ESTADO_MESA[4]:=FALSE;
	IF SERVIR_PLATO1 THEN
		CARGADO1:=FALSE;
	ELSE
		CARGADO2:=FALSE;
	END_IF;
END_IF;

IF (SERVIR_PLATO1 OR SERVIR_PLATO2) AND PS_5 THEN
	ESTADO_MESA[5]:=FALSE;
	IF SERVIR_PLATO1 THEN
		CARGADO1:=FALSE;
	ELSE
		CARGADO2:=FALSE;
	END_IF;
END_IF;

IF (SERVIR_PLATO1 OR SERVIR_PLATO2) AND PS_6 THEN
	ESTADO_MESA[6]:=FALSE;
	IF SERVIR_PLATO1 THEN
		CARGADO1:=FALSE;
	ELSE
		CARGADO2:=FALSE;
	END_IF;
END_IF;

IF (SERVIR_PLATO1 OR SERVIR_PLATO2) AND PS_7 THEN
	ESTADO_MESA[7]:=FALSE;
	IF SERVIR_PLATO1 THEN
		CARGADO1:=FALSE;
	ELSE
		CARGADO2:=FALSE;
	END_IF;
END_IF;

IF (SERVIR_PLATO1 OR SERVIR_PLATO2) AND PS_8 THEN
	ESTADO_MESA[8]:=FALSE;
	IF SERVIR_PLATO1 THEN
		CARGADO1:=FALSE;
	ELSE
		CARGADO2:=FALSE;
	END_IF;
END_IF;
END_PROGRAM

(* POU VIS_PISTON, ST *)
PROGRAM VIS_PISTON
VAR
END_VAR
(*Actuadores piston*)
IF PISCLA_MAS THEN
	pistonx:=pistonx+vpist;
END_IF;
IF PISCLA_MENOS THEN
	pistonx:=pistonx-(vpist*2);
END_IF;



(*Sensores piston*)
IF pistonx<=0 THEN
	FC_PISCLA:=TRUE;
ELSE
	FC_PISCLA:=FALSE;
END_IF;
END_PROGRAM

(* POU VIS_CINTAS_PLATO, ST *)
PROGRAM VIS_CINTAS_PLATO
VAR
	i:INT;
	j:INT := 1;
	fs_disp:BOOL := FALSE;
	F_ENT_COC:BOOL;
	F_ENT_CLA:BOOL;
	F_ENT_H1:BOOL;
	F_ENT_H2:BOOL;
	F_ENT_H3:BOOL;
	F_ENT_SERVIR:BOOL;
	F_ESPERA_H1:BOOL;
	F_ESPERA_H2:BOOL;
	F_ESPERA_H3:BOOL;
	F_S_H1:BOOL;
	F_S_H2:BOOL;
	F_S_H3:BOOL;
	F_ENT_REAL1:BOOL;
	F_ENT_REAL2:BOOL;
	F_ENT_REAL3:BOOL;
	F_SEM_H2_R:BOOL;
	F_SEM_H2_V:BOOL;
	F_SEM_H1_R:BOOL;
	F_SEM_H1_V:BOOL;
	F_SAL_R:BOOL;
	F_ENT_TER:BOOL;
	F_TER_1:BOOL;
	F_TER_2:BOOL;
	F_TER_3:BOOL;
END_VAR
(*Dispensadora de platos*)
IF DISP_PLATO THEN (*detetor de flanco de subida de DISP_PLATO*)
	IF NOT fs_disp THEN
		plato[j].x:=0;
		plato[j].y:=0;
		plato[j].on:=TRUE;
		fs_disp:=TRUE;
		j:=j+1;
		IF j=9 THEN
		j:=1;
		END_IF;
	END_IF;
ELSE
	fs_disp:=FALSE;
END_IF;

(*ACTUADORES*)
FOR i:=1 TO 8 BY 1 DO
	IF plato[i].on THEN
		(*cinta entrada cocina*)
		IF plato[i].x>=-25 AND plato[i].x<=25 AND plato[i].y>=-30 AND plato[i].y<=200 AND CIN_ENT_COC THEN
			plato[i].y:=plato[i].y+velp;
		END_IF;

		(*cinta clasificador*)
		IF plato[i].x>=-5 AND plato[i].x<=25 AND plato[i].y>=200 AND plato[i].y<=430 AND CIN_CLA THEN
			plato[i].y:=plato[i].y+velp;
		END_IF;

		(*cinta entrada h1*)
		IF CIN_H1 THEN
			IF plato[i].x>=25 AND plato[i].x<=75 AND plato[i].y>=380 AND plato[i].y<=530 AND NOT (plato[i].y>=380 AND plato[i].y<=450 AND plato[i].x>=(-20+pistonx) AND plato[i].x<=pistonx AND AGARRAR)  THEN
				plato[i].y:=plato[i].y+velp;
			END_IF;

			IF plato[i].x>=-205 AND plato[i].x<=75 AND plato[i].y>=510 AND plato[i].y<=555 THEN
				plato[i].x:=plato[i].x-velp;
			END_IF;

			IF plato[i].x>=-220 AND plato[i].x<=-205 AND plato[i].y>=510 AND plato[i].y<=720 THEN
				plato[i].y:=plato[i].y+velp;
			END_IF;
		END_IF;

		(*cinta entrada h2*)
		IF plato[i].x>=75 AND plato[i].x<=125 AND plato[i].y>=380 AND plato[i].y<=720 AND CIN_H2 AND NOT(plato[i].y>=380 AND plato[i].y<=450 AND plato[i].x>=(-20+pistonx) AND plato[i].x<=pistonx AND AGARRAR)  THEN
			plato[i].y:=plato[i].y+velp;
		END_IF;

		(*cinta entrada h3*)
		IF CIN_H3 THEN
			IF plato[i].x>=125 AND plato[i].x<=175 AND plato[i].y>=380 AND plato[i].y<=530 AND NOT (plato[i].y>=380 AND plato[i].y<=450 AND plato[i].x>=(-20+pistonx) AND plato[i].x<=pistonx AND AGARRAR)  THEN
				plato[i].y:=plato[i].y+velp;
			END_IF;

			IF plato[i].x>=125 AND plato[i].x<=410 AND plato[i].y>=510 AND plato[i].y<=555 THEN
				plato[i].x:=plato[i].x+velp;
			END_IF;

			IF plato[i].x>=405 AND plato[i].x<=440 AND plato[i].y>=510 AND plato[i].y<=720 THEN
				plato[i].y:=plato[i].y+velp;
			END_IF;
		END_IF;

		(*cinta salida h1*)
		IF plato[i].x>=-235 AND plato[i].x<=-185 AND plato[i].y>=715 AND plato[i].y<=870 AND CIN_H1_A_REAL THEN
			plato[i].y:=plato[i].y+velp;
		END_IF;

		(*cinta salida h2*)
		IF plato[i].x>=75 AND plato[i].x<=125 AND plato[i].y>=715 AND plato[i].y<=870 AND CIN_H2_A_REAL THEN
			plato[i].y:=plato[i].y+velp;
		END_IF;

		(*cinta salida h3*)
		IF plato[i].x>=405 AND plato[i].x<=435 AND plato[i].y>=715 AND plato[i].y<=870 AND CIN_H3_A_REAL THEN
			plato[i].y:=plato[i].y+velp;
		END_IF;

		(*cinta realimentacion*)
		IF CIN_REALIM THEN
			IF plato[i].x>=-415 AND plato[i].x<=435 AND plato[i].y>=870 AND plato[i].y<=895 THEN
				plato[i].x:=plato[i].x-velp;
			END_IF;

			IF plato[i].x>=-445 AND plato[i].x<=-410 AND plato[i].y>=230 AND plato[i].y<=895 THEN
				plato[i].y:=plato[i].y-velp;
			END_IF;

			IF plato[i].x>=-445 AND plato[i].x<0 AND plato[i].y>=205 AND plato[i].y<=235 THEN
				plato[i].x:=plato[i].x+velp;
			END_IF;
		END_IF;

		(*cinta servicio a mesa*)
		IF CIN_SERVIR AND NOT (plato[i].y>=380 AND plato[i].y<=450 AND plato[i].x>=(-20+pistonx) AND plato[i].x<=pistonx AND AGARRAR)  THEN
			IF plato[i].x>=175 AND plato[i].x<=510 AND plato[i].y>=385 AND plato[i].y<=435 THEN
				plato[i].x:=plato[i].x+velp;
			END_IF;

			IF plato[i].x>=505 AND plato[i].x<=535 AND plato[i].y>=205 AND plato[i].y<=435 THEN
				plato[i].y:=plato[i].y-velp;
			END_IF;
		END_IF;

		(*Cinta cola mesa*)
		IF plato[i].x>=475 AND plato[i].x<=535 AND plato[i].y>=-115 AND plato[i].y<=205 AND CIN_COLA_SERV THEN
			plato[i].y:=plato[i].y-velp;
		END_IF;

		(*movimiento piston*)
		IF plato[i].y>=385 AND plato[i].y<=445 AND plato[i].x>=(-15+pistonx) AND plato[i].x<=(-10+pistonx) THEN
			plato[i].x:=plato[i].x+vpist;
		END_IF;

		(*servir*)
		IF plato[i].x>=475 AND plato[i].x<=570 AND plato[i].y > 150 AND plato[i].y <= 170 AND CARGAR_PLATO[1] THEN
			plato[i].x:=plato[i].x+9;
		END_IF;
		IF plato[i].x>=565 AND plato[i].x<=585 AND plato[i].y > 150 AND plato[i].y <= 170 THEN
			plato[i].on:=FALSE;
			IF PR1_1 THEN
				CARGADO1:=TRUE;
			ELSIF PR2_1 THEN
				CARGADO2:=TRUE;
			END_IF;
		END_IF;

		IF plato[i].x>=475 AND plato[i].x<=570 AND plato[i].y > 30 AND plato[i].y <= 50 AND CARGAR_PLATO[2] THEN
			plato[i].x:=plato[i].x+9;
		END_IF;
		IF plato[i].x>=565 AND plato[i].x<=585 AND plato[i].y > 30 AND plato[i].y <= 50 THEN
			plato[i].on:=FALSE;
			IF PR1_2 THEN
				CARGADO1:=TRUE;
			ELSIF PR2_2 THEN
				CARGADO2:=TRUE;
			END_IF;
		END_IF;

		IF plato[i].x>=475 AND plato[i].x<=570 AND plato[i].y > -85 AND plato[i].y <= -75 AND CARGAR_PLATO[3] THEN
			plato[i].x:=plato[i].x+9;
		END_IF;
		IF plato[i].x>=565 AND plato[i].x<=585 AND plato[i].y > -85 AND plato[i].y <= -75 THEN
			plato[i].on:=FALSE;
			IF PR1_3 THEN
				CARGADO1:=TRUE;
			ELSIF PR2_3 THEN
				CARGADO2:=TRUE;
			END_IF;
		END_IF;

	END_IF;
END_FOR;


(*SENSORES*)
F_ENT_COC:=FALSE;
F_ENT_CLA:=FALSE;
F_ENT_H1:=FALSE;
F_ENT_H2:=FALSE;
F_ENT_H3:=FALSE;
F_ENT_REAL1:=FALSE;
F_ENT_REAL2:=FALSE;
F_ENT_REAL3:=FALSE;
F_ENT_SERVIR:=FALSE;
F_ENT_TER:=FALSE;
F_ESPERA_H1:=FALSE;
F_ESPERA_H2:=FALSE;
F_ESPERA_H3:=FALSE;
F_S_H1:=FALSE;
F_S_H2:=FALSE;
F_S_H3:=FALSE;
F_SAL_R:=FALSE;
F_SEM_H1_R:=FALSE;
F_SEM_H1_V:=FALSE;
F_SEM_H2_R:=FALSE;
F_SEM_H2_V:=FALSE;
F_TER_1:=FALSE;
F_TER_2:=FALSE;
F_TER_3:=FALSE;

FOR i:=1 TO 8 BY 1 DO
	IF plato[i].on THEN
		IF plato[i].x>=-25 AND plato[i].x <=25 AND plato[i].y >= 165 AND plato[i].y <= 210 THEN
			F_ENT_COC:=TRUE;
		END_IF;

		IF plato[i].x>=-25 AND plato[i].x <=25 AND plato[i].y >= 255 AND plato[i].y <= 290 THEN
			S_CLA[i]:=TRUE;
		ELSE
			S_CLA[i]:=FALSE;
		END_IF;

		IF plato[i].x>=-25 AND plato[i].x <=25 AND plato[i].y >= 405 AND plato[i].y <= 420 THEN
			F_ENT_CLA:=TRUE;
		END_IF;

		IF plato[i].x>45 AND plato[i].x <=75 AND plato[i].y >= 405 AND plato[i].y <= 420 THEN
			F_ENT_H1:=TRUE;
		END_IF;

		IF plato[i].x>95 AND plato[i].x <=125 AND plato[i].y >= 405 AND plato[i].y <= 420 THEN
			F_ENT_H2:=TRUE;
		END_IF;

		IF plato[i].x>145 AND plato[i].x <=175 AND plato[i].y >= 405 AND plato[i].y <= 420 THEN
			F_ENT_H3:=TRUE;
		END_IF;

		IF plato[i].x>195 AND plato[i].x <=225 AND plato[i].y >= 405 AND plato[i].y <= 420 THEN
			F_ENT_SERVIR:=TRUE;
		END_IF;

		IF plato[i].x>-220 AND plato[i].x <=-205 AND plato[i].y >= 635 AND plato[i].y <= 680 THEN
			F_ESPERA_H1:=TRUE;
		END_IF;

		IF plato[i].x>75 AND plato[i].x <=125 AND plato[i].y >= 635 AND plato[i].y <= 680 THEN
			F_ESPERA_H2:=TRUE;
		END_IF;

		IF plato[i].x>405 AND plato[i].x <=440 AND plato[i].y >= 635 AND plato[i].y <= 680 THEN
			F_ESPERA_H3:=TRUE;
		END_IF;

		IF plato[i].x>-230 AND plato[i].x <=-190 AND plato[i].y >= 720 AND plato[i].y <= 730 THEN
			F_S_H1:=TRUE;
		END_IF;

		IF plato[i].x>80 AND plato[i].x <=120 AND plato[i].y >= 720 AND plato[i].y <= 730 THEN
			F_S_H2:=TRUE;
		END_IF;

		IF plato[i].x>390 AND plato[i].x <=430 AND plato[i].y >= 720 AND plato[i].y <= 730 THEN
			F_S_H3:=TRUE;
		END_IF;

		IF plato[i].x>-220 AND plato[i].x <=-205 AND plato[i].y >= 810 AND plato[i].y <= 870 THEN
			F_ENT_REAL1:=TRUE;
		END_IF;

		IF plato[i].x>75 AND plato[i].x <=125 AND plato[i].y >= 810 AND plato[i].y <= 870 THEN
			F_ENT_REAL2:=TRUE;
		END_IF;

		IF plato[i].x>395 AND plato[i].x <=435 AND plato[i].y >= 805 AND plato[i].y <= 870 THEN
			F_ENT_REAL3:=TRUE;
		END_IF;

		IF plato[i].x>125 AND plato[i].x <=180 AND plato[i].y > 840 AND plato[i].y <= 880 THEN
			F_SEM_H2_R:=TRUE;
		END_IF;

		IF plato[i].x>35 AND plato[i].x <=90 AND plato[i].y > 840 AND plato[i].y <= 880 THEN
			F_SEM_H2_V:=TRUE;
		END_IF;

		IF plato[i].x>-175 AND plato[i].x <=-130 AND plato[i].y > 840 AND plato[i].y <= 880 THEN
			F_SEM_H1_R:=TRUE;
		END_IF;

		IF plato[i].x>-265 AND plato[i].x <=-240 AND plato[i].y > 840 AND plato[i].y <= 880 THEN
			F_SEM_H1_V:=TRUE;
		END_IF;

		IF plato[i].x>-90 AND plato[i].x <=-70 AND plato[i].y >200 AND plato[i].y <= 240 THEN
			F_SAL_R:=TRUE;
		END_IF;

		IF plato[i].x>480 AND plato[i].x <=530 AND plato[i].y > 275 AND plato[i].y <= 285 THEN
			F_ENT_TER:=TRUE;
		END_IF;

		IF plato[i].x>480 AND plato[i].x <=530 AND plato[i].y > 155 AND plato[i].y <= 165 THEN
			F_TER_1:=TRUE;
		END_IF;

		IF plato[i].x>480 AND plato[i].x <530 AND plato[i].y > 35 AND plato[i].y <= 45 THEN
			F_TER_2:=TRUE;
		END_IF;

		IF plato[i].x>480 AND plato[i].x <=530 AND plato[i].y > -85 AND plato[i].y <= -75 THEN
			F_TER_3:=TRUE;
		END_IF;

	END_IF;
END_FOR;

IF F_ENT_COC THEN
	ENT_COC:=TRUE;
ELSE
	ENT_COC:=FALSE;
END_IF;

IF F_ENT_CLA THEN
	ENT_CLA:=TRUE;
ELSE
	ENT_CLA:=FALSE;
END_IF;

IF F_ENT_H1 THEN
	ENT_H1:=TRUE;
ELSE
	ENT_H1:=FALSE;
END_IF;

IF F_ENT_H2 THEN
	ENT_H2:=TRUE;
ELSE
	ENT_H2:=FALSE;
END_IF;

IF F_ENT_H3 THEN
	ENT_H3:=TRUE;
ELSE
	ENT_H3:=FALSE;
END_IF;

IF F_ENT_REAL1 THEN
	ENT_REAL1:=TRUE;
ELSE
	ENT_REAL1:=FALSE;
END_IF;

IF F_ENT_REAL2 THEN
	ENT_REAL2:=TRUE;
ELSE
	ENT_REAL2:=FALSE;
END_IF;

IF F_ENT_REAL3 THEN
	ENT_REAL3:=TRUE;
ELSE
	ENT_REAL3:=FALSE;
END_IF;

IF F_ENT_SERVIR THEN
	ENT_SERVIR:=TRUE;
ELSE
	ENT_SERVIR:=FALSE;
END_IF;

IF F_ENT_TER THEN
	ENT_TER:=TRUE;
ELSE
	ENT_TER:=FALSE;
END_IF;

IF F_ESPERA_H1 THEN
	ESPERA_H1:=TRUE;
ELSE
	ESPERA_H1:=FALSE;
END_IF;

IF F_ESPERA_H2 THEN
	ESPERA_H2:=TRUE;
ELSE
	ESPERA_H2:=FALSE;
END_IF;

IF F_ESPERA_H3 THEN
	ESPERA_H3:=TRUE;
ELSE
	ESPERA_H3:=FALSE;
END_IF;

IF F_S_H1 THEN
	S_H1:=TRUE;
ELSE
	S_H1:=FALSE;
END_IF;

IF F_S_H2 THEN
	S_H2:=TRUE;
ELSE
	S_H2:=FALSE;
END_IF;

IF F_S_H3 THEN
	S_H3:=TRUE;
ELSE
	S_H3:=FALSE;
END_IF;

IF F_SAL_R THEN
	SAL_R:=TRUE;
ELSE
	SAL_R:=FALSE;
END_IF;

IF F_SEM_H1_R THEN
	SEM_H1_R:=TRUE;
ELSE
	SEM_H1_R:=FALSE;
END_IF;

IF F_SEM_H1_V THEN
	SEM_H1_V:=TRUE;
ELSE
	SEM_H1_V:=FALSE;
END_IF;

IF F_SEM_H2_R THEN
	SEM_H2_R:=TRUE;
ELSE
	SEM_H2_R:=FALSE;
END_IF;

IF F_SEM_H2_V THEN
	SEM_H2_V:=TRUE;
ELSE
	SEM_H2_V:=FALSE;
END_IF;

IF F_TER_1 THEN
	TER_1:=TRUE;
ELSE
	TER_1:=FALSE;
END_IF;

IF F_TER_2 THEN
	TER_2:=TRUE;
ELSE
	TER_2:=FALSE;
END_IF;

IF F_TER_3 THEN
	TER_3:=TRUE;
ELSE
	TER_3:=FALSE;
END_IF;
END_PROGRAM

(* POU VIS_AGV, ST *)
PROGRAM VIS_AGV
VAR
	incy1: INT;
	incx1: INT;
	v1: INT:=6;
	incy2: INT;
	incx2: INT;
END_VAR
IF MARCHA1=TRUE THEN
	incy1:=0;
	incx1:=0;
	IF y1>=-10 AND y1<=740 AND x1>-20 AND x1<20 THEN (*1 TRAMO*)
		IF y1>=735 AND y1<=747 THEN (*ESQUINA*)
			y1:=740;
		ELSIF y1>=85 AND y1<=95 AND y1<>90 THEN
 (*SENSOR PR_3*)
			y1:=90;
		ELSIF y1>=205 AND y1<=215 AND y1<>210 THEN
 (*SENSOR PR_2*)
			y1:=210;
		ELSIF y1>=325 AND y1<=335 AND y1<>330 THEN
 (*SENSOR PR_1*)
			y1:=330;
		ELSE
			y1:=y1+v1;
		END_IF
	END_IF

	IF x1>=0 AND  x1<=1300 AND y1>730 AND y1<750 THEN(*2 TRAMO*)
		IF x1>=1293 AND x1<=1305 THEN (*ESQUINA*)
			x1:=1300;
		ELSIF x1>75 AND x1<86 AND x1<>80 THEN (*SENSOR BIF_12*)
			x1:=80;
		ELSIF x1>387 AND x1<375 AND x1<>380 THEN (*SENSOR BIF_34*)
			x1:=380;
		ELSIF x1>687 AND x1<674 AND x1<>680 THEN (*SENSOR BIF_56*)
			x1:=680;
		ELSIF x1>981 AND x1<975 AND x1<>980 THEN (*SENSOR BIF_78*)
			x1:=980;
		ELSE
			x1:=x1+v1;
		END_IF;
	END_IF

	IF y1>290 AND y1<745 AND x1>1299 AND x1<1339 THEN(*3 TRAMO*)
		IF y1>=283 AND y1<= 297 THEN (*ESQUINA*)
			y1:=290;
		ELSE
		y1:=y1-v1;
		END_IF;

	END_IF

	IF x1>460 AND x1<=1319 AND y1>251 AND y1<291 THEN (*4 TRAMO*)
		IF x1>=445 AND x1<=475 THEN (*ESQUINA*)
			x1:=460;
		ELSE
			x1:=x1-v1;
		END_IF;
	END_IF

	IF y1<=290 AND y1>=-20 AND x1<480 AND x1>=440  THEN (*5 TRAMO*)
		IF y1>=-25 AND y1<=15 THEN (*ESQUINA*)
			y1:=0;
		ELSE
			y1:=y1-v1;
		END_IF
	END_IF

	IF x1<=460 AND x1>0 AND y1<19 AND y1>-29  THEN (*6 TRAMO*)
		IF x1>=-5 AND x1<=7 THEN (*ESQUINA*)
			x1:=0;
		ELSIF x1>125 AND x1<135 AND x1<>130 THEN (*SENSOR PC_1*)
			x1:=130;
		ELSIF x1>327 AND x1<333 AND x1<>330 THEN (*SENSOR PC_2*)
			x1:=330;
		ELSE
			x1:=x1-v1;
		END_IF;
	END_IF
END_IF

IF MARCHA2=TRUE THEN
	incy2:=0;
	incx2:=0;
	IF y2>=0 AND y2<=740 AND x2>-20 AND x2<20 THEN
		y2:=y2+v1;
	END_IF

	IF x2>=0 AND  x2<=1300 AND y2>730 AND y2<750THEN
		x2:=x2+v1;
	END_IF

	IF y2>290 AND y2<745 AND x2>1299 AND x2<1339 THEN
		y2:=y2-v1;
	END_IF

	IF x2>460 AND x2<=1319 AND y2>251 AND y2<291 THEN
		x2:=x2-v1;
	END_IF

	IF y2<=290 AND y2>=-20 AND x2<480 AND x2>440  THEN
		y2:=y2-v1;
	END_IF

	IF x2<=460 AND x2>0 AND y2<19 AND y2>-29  THEN
		x2:=x2-v1;
	END_IF
END_IF

(*BIFURCACION HACIA  ARRIBA*)

IF BIF_ARRIBA1=TRUE THEN
	IF incy1>=0 AND incy1<310 AND incx1=0 THEN (*TRAMO 1*)
		IF incy1>=306 AND incy1<315 AND incy1<>310 THEN (*ESQUINA Y*)
			incy1:=310;
		ELSE
		y1:=y1-v1;
		incy1:=incy1+v1;
		END_IF

	END_IF;

	IF incy1>=310 AND incx1>=0 AND incx1<=240 THEN (*TRAMO 2*)
		IF incx1>195 AND incx1<207 AND incx1<>200 THEN (*SENSOR PS_X*)
			incx1:=200;
		ELSIF incx1>237 AND incx1<246 AND incx1<>240  THEN (*ESQUINA  X*)
			incx1:=240;
		END_IF
		x1:=x1+v1;
		incx1:=incx1+v1;
	END_IF;

	IF incy1>=310 AND incy1<=620 AND incx1>=240 THEN (*TRAMO 3*)
END_IF
		IF incy1>513 AND incy1<525 AND incy1<>520 THEN (*SENSOR SS_PS_X*)
			incy1:=520;
		ELSE
			y1:=y1+v1;
			incy1:=incy1+v1;
		END_IF
	END_IF
END_IF

IF BIF_ARRIBA2=TRUE THEN
	IF incy2>=0 AND incy2<310 AND incx2=0 THEN
		y2:=y2-v1;
		incy2:=incy2+v1;
	END_IF;

	IF incy2>=310 AND incx2>=0 AND incx2<=240 THEN
		x2:=x2+v1;
		incx2:=incx2+v1;
	END_IF;

	IF incy2>=310 AND incy2<=620 AND incx2>=240 THEN
		y2:=y2+v1;
		incy2:=incy2+v1;
	END_IF
END_IF

(*BIFURCACION HACIA  ABAJO*)
IF BIF_ABAJO1=TRUE THEN
	IF incy1>=0 AND incy1<300 AND incx1=0 THEN
		y1:=y1+v1;
		incy1:=incy1+v1;
	END_IF

	IF incy1>=300 AND incx1>=0 AND incx1<=240 THEN
		x1:=x1+v1;
		incx1:=incx1+v1;
	END_IF

	IF incy1>=300 AND incy1<=600 AND incx1>=240 THEN
		y1:=y1-v1;
		incy1:=incy1+v1;
	END_IF
END_IF

IF BIF_ABAJO2=TRUE THEN
	IF incy2>=0 AND incy2<300 AND incx2=0 THEN
		y2:=y2+v1;
		incy2:=incy2+v1;
	END_IF

	IF incy2>=300 AND incx2>=0 AND incx2<=240 THEN
		x2:=x2+v1;
		incx2:=incx2+v1;
	END_IF

	IF incy2>=300 AND incy2<=600 AND incx2>=240 THEN
		y2:=y2-v1;
		incy2:=incy2+v1;
	END_IF
END_IF



(*SENSORES*)

IF x1>=128  AND x1<=132   AND y1>=-2   AND y1<=2 THEN
	PC1_1:=TRUE;
ELSE
	PC1_1:=FALSE;
END_IF
IF x1>=328  AND x1<332   AND y1>=-2   AND y1<=2 THEN
	PC1_2:=TRUE;
ELSE
	PC1_2:=FALSE;
END_IF
IF x1>=-2  AND x1<=2   AND y1>=88   AND y1<=92 THEN
	PR1_3:=TRUE;
ELSE
	PR1_3:=FALSE;
END_IF
IF x1>=-2  AND x1<=2   AND y1>=208   AND y1<=212 THEN
	PR1_2:=TRUE;
ELSE
	PR1_2:=FALSE;
END_IF
IF x1>=-2  AND x1<=2   AND y1>=328   AND y1<=332 THEN
	PR1_1:=TRUE;
ELSE
	PR1_1:=FALSE;
END_IF
IF x1>=78  AND x1<=82   AND y1>=730   AND y1<=750 THEN
	BIF1_12:=TRUE;
ELSE
	BIF1_12:=FALSE;
END_IF
IF x1>=378  AND x1<=382   AND y1>=730   AND y1<=750 THEN
	BIF1_34:=TRUE;
ELSE
	BIF1_34:=FALSE;
END_IF
IF x1>=678  AND x1<=682   AND y1>=730   AND y1<=750 THEN
	BIF1_56:=TRUE;
ELSE
	BIF1_56:=FALSE;
END_IF
IF x1>=978  AND x1<=982   AND y1>=730   AND y1<=750 THEN
	BIF1_78:=TRUE;
ELSE
	BIF1_78:=FALSE;
END_IF



IF x2>=128  AND x2<=132   AND y2>=-2   AND y2<=2 THEN
	PC2_1:=TRUE;
ELSE
	PC2_1:=FALSE;
END_IF
IF x2>=328  AND x2<332   AND y2>=-2   AND y2<=2 THEN
	PC2_2:=TRUE;
ELSE
	PC2_2:=FALSE;
END_IF
IF x2>=-2  AND x2<=2   AND y2>=88   AND y2<=92 THEN
	PR2_3:=TRUE;
ELSE
	PR2_3:=FALSE;
END_IF
IF x2>=-2  AND x2<=2   AND y2>=208   AND y2<=212 THEN
	PR2_2:=TRUE;
ELSE
	PR2_2:=FALSE;
END_IF
IF x2>=-2  AND x2<=2   AND y2>=328   AND y2<=332 THEN
	PR2_1:=TRUE;
ELSE
	PR2_1:=FALSE;
END_IF
IF x2>=78  AND x2<=82   AND y2>=730   AND y2<=750 THEN
	BIF2_12:=TRUE;
ELSE
	BIF2_12:=FALSE;
END_IF
IF x2>=378  AND x2<=382   AND y2>=730   AND y2<=750 THEN
	BIF2_34:=TRUE;
ELSE
	BIF2_34:=FALSE;
END_IF
IF x2>=678  AND x2<=682   AND y2>=730   AND y2<=750 THEN
	BIF2_56:=TRUE;
ELSE
	BIF2_56:=FALSE;
END_IF
IF x2>=978  AND x2<=982   AND y2>=730   AND y2<=750 THEN
	BIF2_78:=TRUE;
ELSE
	BIF2_78:=FALSE;
END_IF



IF (x1>=198 AND x1<=202 AND y1>=420 AND y1<=440) OR (x2>=198 AND x2<=202 AND y2>=420 AND y2<=440) THEN
	PS_1:=TRUE;
ELSE
	PS_1:=FALSE;
END_IF
IF (x1>=198 AND x1<=202 AND y1>=1030 AND y1<=1050) OR (x2>=198 AND x2<=202 AND y2>=1030 AND y2<=1050) THEN
	PS_2:=TRUE;
ELSE
	PS_2:=FALSE;
END_IF
IF (x1>=498 AND x1<=502 AND y1>=420 AND y1<=440) OR (x2>=498 AND x2<502 AND y2>=420 AND y2<=440) THEN
	PS_3:=TRUE;
ELSE
	PS_3:=FALSE;
END_IF
IF (x1>=498 AND x1<=502 AND y1>=1030 AND y1<=1050) OR (x2>=498 AND x2<=502 AND y2>=1030 AND y2<=1050) THEN
	PS_4:=TRUE;
ELSE
	PS_4:=FALSE;
END_IF
IF (x1>=798 AND x1<=802 AND y1>=420 AND y1<=440) OR (x2>=798 AND x2<=802 AND y2>=420 AND y2<=440) THEN
	PS_5:=TRUE;
ELSE
	PS_5:=FALSE;
END_IF
IF (x1>=798 AND x1<=802 AND y1>=1030 AND y1<=1050) OR (x2>=798 AND x2<=802 AND y2>=1030 AND y2<=1050) THEN
	PS_6:=TRUE;
ELSE
	PS_6:=FALSE;
END_IF
IF (x1>=1098 AND x1<=1102 AND y1>=420 AND y1<=440) OR (x2>=1098 AND x2<=1102 AND y2>=420 AND y2<=440) THEN
	PS_7:=TRUE;
ELSE
	PS_7:=FALSE;
END_IF
IF (x1>=1098 AND x1<=1102 AND y1>=1030 AND y1<=1050) OR (x2>=1098 AND x2<=1102 AND y2>=1030 AND y2<=1050) THEN
	PS_8:=TRUE;
ELSE
	PS_8:=FALSE;
END_IF


IF (x1>=310 AND x1<=330 AND y1>=638 AND y1<=642) OR (x2>=310 AND x2<=330 AND y2>=638 AND y2<=642) THEN
	SS_PS_1:=TRUE;
ELSE
	SS_PS_1:=FALSE;
END_IF
IF (x1>=310 AND x1<=330 AND y1>=828 AND y1<=832) OR (x2>=310 AND x2<=330 AND y2>=828 AND y2<=832) THEN
	SS_PS_2:=TRUE;
ELSE
	SS_PS_2:=FALSE;
END_IF
IF (x1>=610 AND x1<=630 AND y1>=638 AND y1<=642) OR (x2>=610 AND x2<=630 AND y2>=638 AND y2<=642) THEN
	SS_PS_3:=TRUE;
ELSE
	SS_PS_3:=FALSE;
END_IF
IF (x1>=610 AND x1<=630 AND y1>=828 AND y1<=842) OR (x2>=610 AND x2<=630 AND y2>=828 AND y2<=842) THEN
	SS_PS_4:=TRUE;
ELSE
	SS_PS_4:=FALSE;
END_IF
IF (x1>=910 AND x1<=930 AND y1>=638 AND y1<=642) OR (x2>=910 AND x2<=930 AND y2>=638 AND y2<=642) THEN
	SS_PS_5:=TRUE;
ELSE
	SS_PS_5:=FALSE;
END_IF
IF (x1>=910 AND x1<=930 AND y1>=828 AND y1<=832) OR (x2>=910 AND x2<=930 AND y2>=828 AND y2<=832) THEN
	SS_PS_6:=TRUE;
ELSE
	SS_PS_6:=FALSE;
END_IF
IF (x1>=1210 AND x1<=1230 AND y1>=638 AND y1<=642) OR (x2>=1210 AND x2<=1230 AND y2>=638 AND y2<=642) THEN
	SS_PS_7:=TRUE;
ELSE
	SS_PS_7:=FALSE;
END_IF
IF (x1>=1210 AND x1<=1230 AND y1>=828 AND y1<=832) OR (x2>=1210 AND x2<=1230 AND y2>=828 AND y2<=832) THEN
	SS_PS_8:=TRUE;
ELSE
	SS_PS_8:=FALSE;
END_IF
IF (x1>=1290 AND x1<=1310 AND y1>=730 AND y1<=750) OR (x2>=1290 AND x2<=1310 AND y2>=730 AND y2<=750) THEN
	SS_F:=TRUE;
ELSE
	SS_F:=FALSE;
END_IF
END_PROGRAM

(* POU COLAS_PEDIDOS, ST *)
PROGRAM COLAS_PEDIDOS
VAR
	FS_PE1:BOOL;
	FS_PE2:BOOL;
	FS_PE3:BOOL;
	FS_M1:BOOL;
	FS_M2:BOOL;
	FS_M3:BOOL;
	FS_M4:BOOL;
	FS_M5:BOOL;
	FS_M6:BOOL;
	FS_M7:BOOL;
	FS_M8:BOOL;
	FLAG_PE:BOOL;
	i: INT;
	FLAG_MP: BOOL;
	i_pedido_temp:INT;
	i_pedidomesa_temp:INT;
END_VAR
(******************************************************PEDIDOS***************************************************************)

IF PEDIDO1 AND FS_PE1=FALSE THEN
	FS_PE1:=TRUE;
	B_PEDIDO[1]:=TRUE;
	FOR i:=1 TO 20 BY 1 DO
		IF PENDIENTES_ENTRAR[i]=0 AND FLAG_PE=FALSE THEN
			i_pedido_temp:=i;
			FLAG_PE:=TRUE;
		END_IF
		IF MESA_PEDIDO[i,2]=0 AND FLAG_MP=FALSE THEN
			i_pedidomesa_temp:=i;
			FLAG_MP:=TRUE;
		END_IF
	END_FOR
	FLAG_PE:=FALSE;
	FLAG_MP:=FALSE;
ELSIF PEDIDO1=FALSE THEN
	FS_PE1:=FALSE;
END_IF

IF PEDIDO2 AND FS_PE2=FALSE THEN
	FS_PE2:=TRUE;
	B_PEDIDO[2]:=TRUE;
	FOR i:=1 TO 20 BY 1 DO
		IF PENDIENTES_ENTRAR[i]=0 AND FLAG_PE=FALSE THEN
			i_pedido_temp:=i;
			FLAG_PE:=TRUE;
		END_IF
		IF MESA_PEDIDO[i,2]=0 AND FLAG_MP=FALSE THEN
			i_pedidomesa_temp:=i;
			FLAG_MP:=TRUE;
		END_IF
	END_FOR
	FLAG_PE:=FALSE;
	FLAG_MP:=FALSE;
ELSIF PEDIDO2=FALSE THEN
	FS_PE2:=FALSE;
END_IF

IF PEDIDO3 AND FS_PE3=FALSE THEN
	FS_PE3:=TRUE;
	B_PEDIDO[3]:=TRUE;
	FOR i:=1 TO 20 BY 1 DO
		IF PENDIENTES_ENTRAR[i]=0 AND FLAG_PE=FALSE THEN
			i_pedido_temp:=i;
			FLAG_PE:=TRUE;
		END_IF
		IF MESA_PEDIDO[i,2]=0 AND FLAG_MP=FALSE THEN
			i_pedidomesa_temp:=i;
			FLAG_MP:=TRUE;
		END_IF
	END_FOR
	FLAG_PE:=FALSE;
	FLAG_MP:=FALSE;
ELSIF PEDIDO3=FALSE THEN
	FS_PE3:=FALSE;
END_IF


(********************************************************MESAS************************************************************)

IF MESA1 AND FS_M1=FALSE THEN
	FS_M1:=TRUE;
	B_MESA[1]:=TRUE;
ELSIF MESA1=FALSE THEN
	FS_M1:=FALSE;
END_IF

IF MESA2 AND FS_M2=FALSE THEN
	FS_M2:=TRUE;
	B_MESA[2]:=TRUE;
ELSIF MESA2=FALSE THEN
	FS_M2:=FALSE;
END_IF

IF MESA3 AND FS_M3=FALSE THEN
	FS_M3:=TRUE;
	B_MESA[3]:=TRUE;
ELSIF MESA3=FALSE THEN
	FS_M3:=FALSE;
END_IF

IF MESA4 AND FS_M4=FALSE THEN
	FS_M4:=TRUE;
	B_MESA[4]:=TRUE;
ELSIF MESA4=FALSE THEN
	FS_M4:=FALSE;
END_IF

IF MESA5 AND FS_M5=FALSE THEN
	FS_M5:=TRUE;
	B_MESA[5]:=TRUE;
ELSIF MESA5=FALSE THEN
	FS_M5:=FALSE;
END_IF

IF MESA6 AND FS_M6=FALSE THEN
	FS_M6:=TRUE;
	B_MESA[6]:=TRUE;
ELSIF MESA6=FALSE THEN
	FS_M6:=FALSE;
END_IF

IF MESA7 AND FS_M7=FALSE THEN
	FS_M7:=TRUE;
	B_MESA[7]:=TRUE;
ELSIF MESA7=FALSE THEN
	FS_M7:=FALSE;
END_IF

IF MESA8 AND FS_M8=FALSE THEN
	FS_M8:=TRUE;
	B_MESA[8]:=TRUE;
ELSIF MESA8=FALSE THEN
	FS_M8:=FALSE;
END_IF


(******************************CONFIRMACION PEDIDO****************************************)

IF B_PEDIR AND (B_MESA[1] OR B_MESA[2] OR B_MESA[3] OR B_MESA[4] OR B_MESA[5] OR B_MESA[6] OR B_MESA[7] OR B_MESA[8]) AND (B_PEDIDO[1] OR B_PEDIDO[2] OR B_PEDIDO[3]) THEN
	FOR i:=1 TO 3 BY 1 DO
		IF B_PEDIDO[i] THEN
			PENDIENTES_ENTRAR[i_pedido_temp]:=i;
			MESA_PEDIDO[i_pedidomesa_temp,2]:=i;
		END_IF;
		B_PEDIDO[i]:=FALSE;
	END_FOR;

	FOR i:=1 TO 8 BY 1 DO
		IF B_MESA[i] THEN
			MESA_PEDIDO[i_pedidomesa_temp,1]:=i;
		END_IF
		B_MESA[i]:=FALSE;
	END_FOR;
END_IF;

IF B_CANCELAR THEN

	FOR i:=1 TO 3 BY 1 DO
		B_PEDIDO[i]:=FALSE;
	END_FOR;

	FOR i:=1 TO 8 BY 1 DO
		B_MESA[i]:=FALSE;
	END_FOR;

END_IF;
END_PROGRAM

(* Visualisation BOTONERA_AGVS
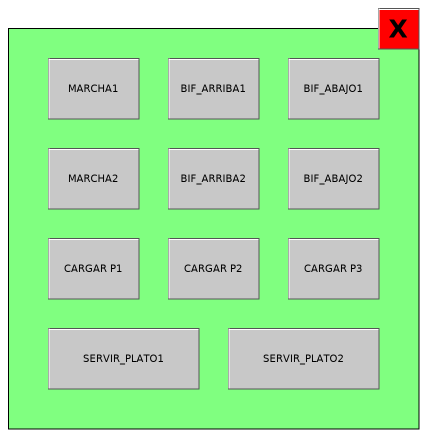
button at (50,70)-(141,131): text "MARCHA1"; toggles .MARCHA1
button at (50,160)-(141,221): text "MARCHA2"; toggles .MARCHA2
button at (170,70)-(261,131): text "BIF_ARRIBA1"; toggles .BIF_ARRIBA1
button at (290,160)-(381,221): text "BIF_ABAJO2"; toggles .BIF_ABAJO2
button at (170,160)-(261,221): text "BIF_ARRIBA2"; toggles .BIF_ARRIBA2
button at (290,70)-(381,131): text "BIF_ABAJO1"; toggles .BIF_ABAJO1
button at (50,250)-(141,311): text "CARGAR P1"; toggles .CARGAR_PLATO[1]
button at (50,340)-(201,401): text "SERVIR_PLATO1"; taps .SERVIR_PLATO1
button at (230,340)-(381,401): text "SERVIR_PLATO2"; taps .SERVIR_PLATO2
button at (170,250)-(261,311): text "CARGAR P2"; toggles .CARGAR_PLATO[2]
button at (290,250)-(381,311): text "CARGAR P3"; toggles .CARGAR_PLATO[3]
button at (380,20)-(421,61): text "X"; opens CONTROL_MANUAL
1 more shapes without text or variables
*)

(* Visualisation BOTONERA_CINTAS
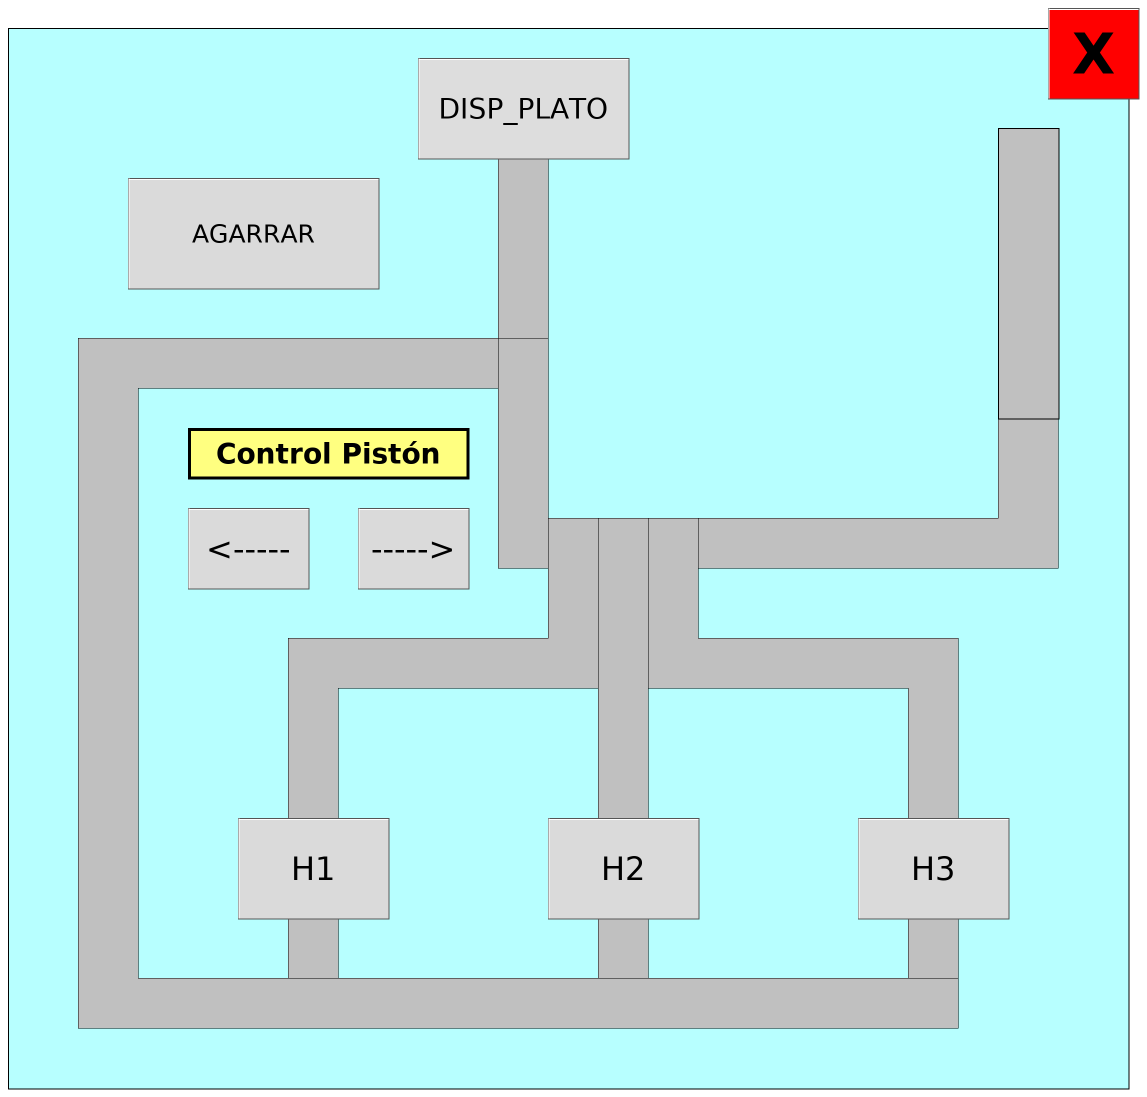
polygon at (640,530)-(690,830): alarm colour if CIN_H2; toggles CIN_H2
polygon at (330,530)-(640,830): alarm colour if CIN_H1; toggles CIN_H1
polygon at (690,530)-(1000,830): alarm colour if CIN_H3; toggles CIN_H3
polygon at (330,930)-(380,990): alarm colour if .CIN_H1_A_REAL; toggles .CIN_H1_A_REAL
polygon at (640,930)-(690,990): alarm colour if .CIN_H2_A_REAL; toggles .CIN_H2_A_REAL
polygon at (950,930)-(1000,990): alarm colour if .CIN_H3_A_REAL; toggles .CIN_H3_A_REAL
polygon at (540,350)-(590,590): alarm colour if CIN_CLA; toggles CIN_CLA
polygon at (120,350)-(1000,1040): alarm colour if .CIN_REALIM; toggles .CIN_REALIM
polygon at (540,120)-(590,360): alarm colour if .CIN_ENT_COC; toggles CIN_ENT_COC
button at (230,520)-(351,601): text "<-----"; taps .PISCLA_MENOS
button at (400,520)-(511,601): text "----->"; taps .PISCLA_MAS
button at (460,70)-(671,171): text "DISP_PLATO"; taps DISP_PLATO
button at (280,830)-(431,931): text "H1"; toggles H1
button at (590,830)-(741,931): text "H2"; toggles H2
button at (900,830)-(1051,931): text "H3"; toggles H3
polygon at (740,430)-(1100,580): alarm colour if .CIN_SERVIR; toggles .CIN_SERVIR
rectangle at (1040,140)-(1101,431): alarm colour if .CIN_COLA_SERV; toggles .CIN_COLA_SERV
rectangle at (230,440)-(511,491): text "Control Pistón"
button at (170,190)-(421,301): text "AGARRAR"; toggles .AGARRAR
button at (1090,20)-(1181,111): text "X"; opens CONTROL_MANUAL
4 more shapes without text or variables
*)

(* Visualisation BOTONERA_PLATOS
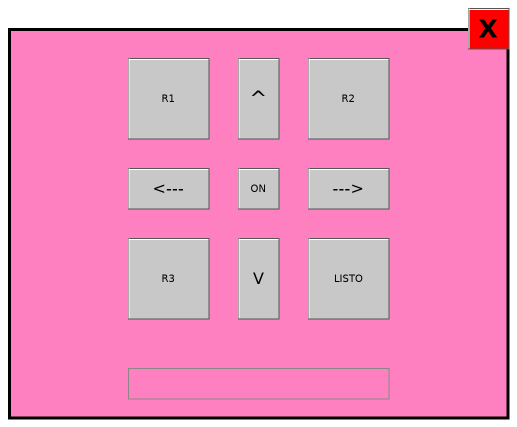
button at (280,60)-(321,141): text "^"; taps bup
button at (350,170)-(431,211): text "--->"; taps bright
button at (170,170)-(251,211): text "<---"; taps bleft
button at (280,240)-(321,321): text "V"; taps bdown
button at (280,170)-(321,211): text "ON"; taps bhide
button at (170,60)-(251,141): text "R1"; taps br1
button at (350,60)-(431,141): text "R2"; taps br2
button at (170,240)-(251,321): text "R3"; taps br3
button at (350,240)-(431,321): text "LISTO"; taps blisto
button at (510,10)-(551,51): text "X"; opens CONTROL_MANUAL
2 more shapes without text or variables
8 elements of other kinds (tables, trends, ...) not read
*)

(* Visualisation CONTROL_MANUAL
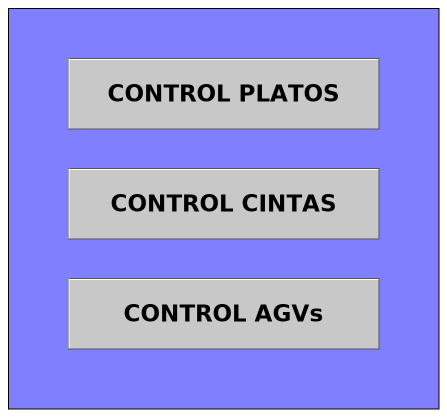
button at (60,50)-(371,121): text "CONTROL PLATOS"; opens BOTONERA_PLATOS
button at (60,160)-(371,231): text "CONTROL CINTAS"; opens BOTONERA_CINTAS
button at (60,270)-(371,341): text "CONTROL AGVs"; opens BOTONERA_AGVS
1 more shapes without text or variables
*)

(* Visualisation VISUAL_RESTAURANTE
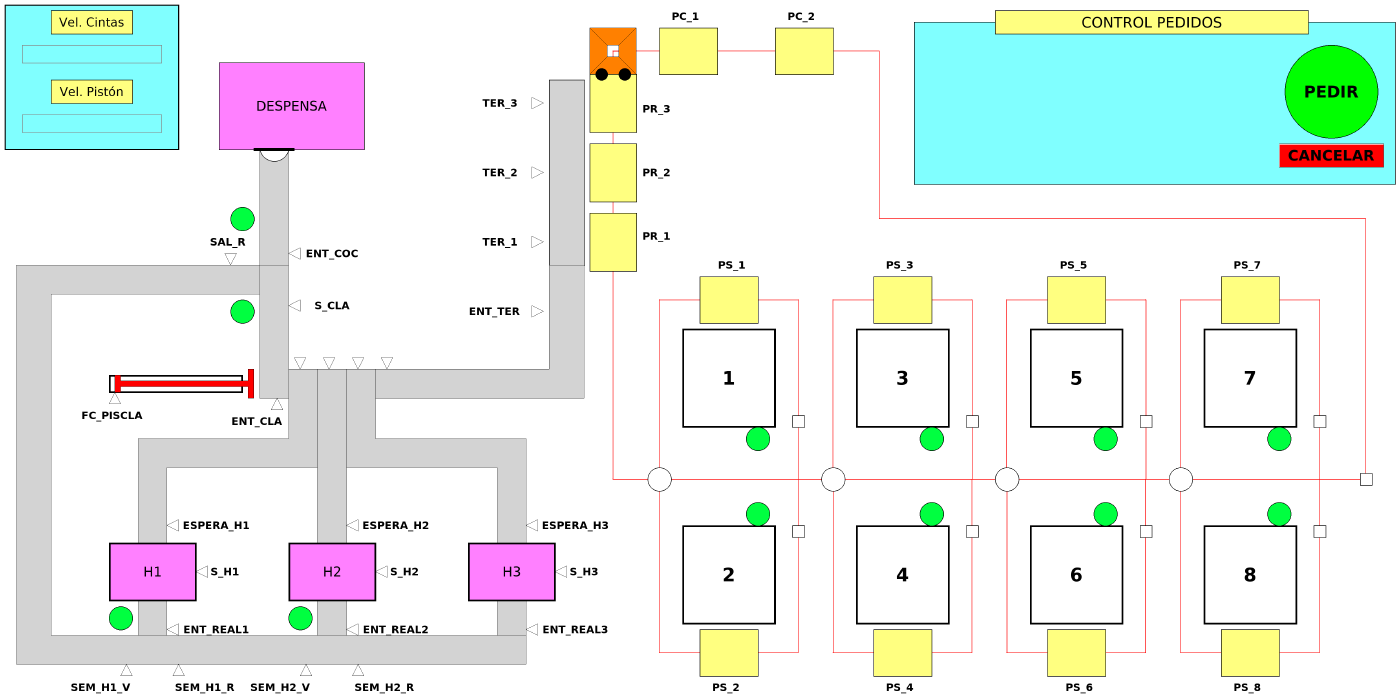
ellipse at (530,250)-(581,301): text "%s"; shows plato[1].receta; invisible if NOT plato[1].on; alarm colour if plato[1].listo; x offset plato[1].x; y offset plato[1].y
polygon at (680,1100)-(700,1120): alarm colour if .ENT_REAL2
polygon at (370,1100)-(390,1120): alarm colour if .ENT_REAL1
polygon at (990,1100)-(1010,1120): alarm colour if .ENT_REAL3
polygon at (690,1170)-(710,1190): alarm colour if .SEM_H2_R
polygon at (380,1170)-(400,1190): alarm colour if .SEM_H1_R
polygon at (600,1170)-(620,1190): alarm colour if .SEM_H2_V
polygon at (290,1170)-(310,1190): alarm colour if .SEM_H1_V
polygon at (270,700)-(290,720): alarm colour if .FC_PISCLA
polygon at (640,640)-(660,660): alarm colour if .ENT_H2
polygon at (690,640)-(710,660): alarm colour if .ENT_H3
polygon at (590,640)-(610,660): alarm colour if .ENT_H1
polygon at (740,640)-(760,660): alarm colour if .ENT_SERVIR
polygon at (470,460)-(490,480): alarm colour if .SAL_R
polygon at (580,450)-(600,470): alarm colour if ENT_COC
polygon at (580,540)-(600,560): alarm colour if .S_CLA[1] OR .S_CLA[2] OR .S_CLA[3]  OR .S_CLA[4]  OR .S_CLA[5]  OR .S_CLA[6]  OR .S_CLA[7]  OR .S_CLA[8]
polygon at (370,920)-(390,940): alarm colour if .ESPERA_H1
polygon at (680,920)-(700,940): alarm colour if .ESPERA_H2
polygon at (990,920)-(1010,940): alarm colour if .ESPERA_H3
polygon at (550,710)-(570,730): alarm colour if .ENT_CLA
polygon at (1000,430)-(1020,450): alarm colour if .TER_1
polygon at (1000,310)-(1020,330): alarm colour if .TER_2
polygon at (1000,190)-(1020,210): alarm colour if .TER_3
polygon at (1000,550)-(1020,570): alarm colour if .ENT_TER
rectangle at (590,440)-(721,481): text "ENT_COC"
rectangle at (610,530)-(701,571): text "S_CLA"
rectangle at (410,420)-(541,461): text "SAL_R"
rectangle at (390,910)-(521,951): text "ESPERA_H1"
rectangle at (700,910)-(831,951): text "ESPERA_H2"
rectangle at (1010,910)-(1141,951): text "ESPERA_H3"
rectangle at (390,1090)-(521,1131): text "ENT_REAL1"
rectangle at (700,1090)-(831,1131): text "ENT_REAL2"
rectangle at (1010,1090)-(1141,1131): text "ENT_REAL3"
rectangle at (210,720)-(341,761): text "FC_PISCLA"
rectangle at (460,730)-(591,771): text "ENT_CLA"
rectangle at (370,1190)-(501,1231): text "SEM_H1_R"
rectangle at (190,1190)-(321,1231): text "SEM_H1_V"
rectangle at (680,1190)-(811,1231): text "SEM_H2_R"
rectangle at (500,1190)-(631,1231): text "SEM_H2_V"
rectangle at (890,180)-(1001,221): text "TER_3"
rectangle at (890,300)-(1001,341): text "TER_2"
rectangle at (890,420)-(1001,461): text "TER_1"
rectangle at (880,540)-(991,581): text "ENT_TER"
rectangle at (430,990)-(511,1031): text "S_H1"
polygon at (420,1000)-(440,1020): alarm colour if .S_H1
rectangle at (740,990)-(821,1031): text "S_H2"
polygon at (730,1000)-(750,1020): alarm colour if .S_H2
rectangle at (1050,990)-(1131,1031): text "S_H3"
polygon at (1040,1000)-(1060,1020): alarm colour if .S_H3
rectangle at (1270,1190)-(1401,1231): text "PS_2"
rectangle at (1570,1190)-(1701,1231): text "PS_4"
rectangle at (1880,1190)-(2011,1231): text "PS_6"
rectangle at (2170,1190)-(2301,1231): text "PS_8"
ellipse at (2100,830)-(2141,871): alarm colour if .BIF1_78 OR .BIF2_78
ellipse at (1800,830)-(1841,871): alarm colour if .BIF1_56 OR .BIF2_56
ellipse at (1500,830)-(1541,871): alarm colour if .BIF1_34 OR .BIF2_34
ellipse at (1200,830)-(1241,871): alarm colour if .BIF1_12 OR .BIF2_12
rounded rectangle at (1260,590)-(1421,761): text "1"; alarm colour if .ESTADO_MESA[1]
rounded rectangle at (1560,590)-(1721,761): text "3"; alarm colour if .ESTADO_MESA[3]
rounded rectangle at (1860,590)-(2021,761): text "5"; alarm colour if .ESTADO_MESA[5]
rounded rectangle at (2160,590)-(2321,761): text "7"; alarm colour if .ESTADO_MESA[7]
rounded rectangle at (1260,930)-(1421,1101): text "2"; alarm colour if .ESTADO_MESA[2]
rounded rectangle at (1560,930)-(1721,1101): text "4"; alarm colour if .ESTADO_MESA[4]
rounded rectangle at (1860,930)-(2021,1101): text "6"; alarm colour if .ESTADO_MESA[6]
rounded rectangle at (2160,930)-(2321,1101): text "8"; alarm colour if .ESTADO_MESA[8]
rectangle at (1100,150)-(1181,251): alarm colour if .PR1_3 OR .PR2_3
rectangle at (1220,70)-(1321,151): alarm colour if .PC1_1 OR .PC2_1
rectangle at (1420,70)-(1521,151): alarm colour if .PC1_2 OR .PC2_2
rectangle at (1290,500)-(1391,581): alarm colour if .PS_1
rectangle at (1590,500)-(1691,581): alarm colour if .PS_3
rectangle at (1890,500)-(1991,581): alarm colour if .PS_5
rectangle at (2190,500)-(2291,581): alarm colour if .PS_7
rectangle at (1290,1110)-(1391,1191): alarm colour if .PS_2
rectangle at (1590,1110)-(1691,1191): alarm colour if .PS_4
rectangle at (1890,1110)-(1991,1191): alarm colour if .PS_6
rectangle at (2190,1110)-(2291,1191): alarm colour if .PS_8
rectangle at (1100,270)-(1181,371): alarm colour if .PR1_2 OR .PR2_2
rectangle at (1100,390)-(1181,491): alarm colour if .PR1_1 OR .PR2_1
rectangle at (1150,190)-(1281,231): text "PR_3"
rectangle at (1150,300)-(1281,341): text "PR_2"
rectangle at (1150,410)-(1281,451): text "PR_1"
rectangle at (1200,30)-(1331,71): text "PC_1"
rectangle at (1400,30)-(1531,71): text "PC_2"
rectangle at (1280,460)-(1411,501): text "PS_1"
rectangle at (1570,460)-(1701,501): text "PS_3"
rectangle at (1870,460)-(2001,501): text "PS_5"
rectangle at (2170,460)-(2301,501): text "PS_7"
ellipse at (270,1070)-(311,1111): alarm colour if .SEM_H1
ellipse at (580,1070)-(621,1111): alarm colour if .SEM_H2
ellipse at (1370,890)-(1411,931): alarm colour if .SEM_M2
ellipse at (1370,760)-(1411,801): alarm colour if .SEM_M1
ellipse at (1670,760)-(1711,801): alarm colour if .SEM_M3
ellipse at (1670,890)-(1711,931): alarm colour if .SEM_M4
ellipse at (1970,760)-(2011,801): alarm colour if .SEM_M5
ellipse at (1970,890)-(2011,931): alarm colour if .SEM_M6
ellipse at (2270,760)-(2311,801): alarm colour if .SEM_M7
ellipse at (2270,890)-(2311,931): alarm colour if .SEM_M8
ellipse at (2300,100)-(2461,261): text "PEDIR"; alarm colour if .B_PEDIR; taps .B_PEDIR
rounded rectangle at (170,40)-(311,81): text "Vel. Cintas"
rounded rectangle at (170,160)-(311,201): text "Vel. Pistón"
rounded rectangle at (1800,40)-(2341,81): text "CONTROL PEDIDOS"
button at (2290,270)-(2471,311): text "CANCELAR"; invisible if NOT (.B_MESA[1] OR .B_MESA[2] OR .B_MESA[3] OR .B_MESA[4] OR .B_MESA[5] OR .B_MESA[6] OR .B_MESA[7] OR .B_MESA[8] ); taps B_CANCELAR
ellipse at (530,250)-(581,301): text "%s"; shows plato[2].receta; invisible if NOT plato[2].on; alarm colour if plato[2].listo; x offset plato[2].x; y offset plato[2].y
ellipse at (530,250)-(581,301): text "%s"; shows plato[4].receta; invisible if NOT plato[4].on; alarm colour if plato[4].listo; x offset plato[4].x; y offset plato[4].y
ellipse at (530,250)-(581,301): text "%s"; shows plato[7].receta; invisible if NOT plato[7].on; alarm colour if plato[7].listo; x offset plato[7].x; y offset plato[7].y
ellipse at (530,250)-(581,301): text "%s"; shows plato[8].receta; invisible if NOT plato[8].on; alarm colour if plato[8].listo; x offset plato[8].x; y offset plato[8].y
ellipse at (530,250)-(581,301): text "%s"; shows plato[3].receta; invisible if NOT plato[3].on; alarm colour if plato[3].listo; x offset plato[3].x; y offset plato[3].y
ellipse at (530,250)-(581,301): text "%s"; shows plato[5].receta; invisible if NOT plato[5].on; alarm colour if plato[5].listo; x offset plato[5].x; y offset plato[5].y
ellipse at (530,250)-(581,301): text "%s"; shows plato[6].receta; invisible if NOT plato[6].on; alarm colour if plato[6].listo; x offset plato[6].x; y offset plato[6].y
polygon at (280,660)-(520,710): x offset pistonx
rectangle at (270,960)-(421,1061): text "H1"; alarm colour if .H1
rectangle at (580,960)-(731,1061): text "H2"; alarm colour if .H2
rectangle at (890,960)-(1041,1061): text "H3"; alarm colour if .H3
rounded rectangle at (460,130)-(711,281): text "DESPENSA"; alarm colour if .DISP_PLATO
rectangle at (1450,740)-(1471,761): alarm colour if .SS_PS_1
rectangle at (1450,930)-(1471,951): alarm colour if .SS_PS_2
rectangle at (1750,740)-(1771,761): alarm colour if .SS_PS_3
rectangle at (1750,930)-(1771,951): alarm colour if .SS_PS_4
rectangle at (2050,740)-(2071,761): alarm colour if .SS_PS_5
rectangle at (2050,930)-(2071,951): alarm colour if .SS_PS_6
rectangle at (2350,740)-(2371,761): alarm colour if .SS_PS_7
rectangle at (2350,930)-(2371,951): alarm colour if .SS_PS_8
rectangle at (2430,840)-(2451,861): alarm colour if .SS_F
polygon at (1100,70)-(1180,150): alarm colour if CARGADO1; x offset x1; y offset y1
ellipse at (1110,140)-(1131,161): x offset x1; y offset y1
ellipse at (1150,140)-(1171,161): x offset x1; y offset y1
polygon at (1100,70)-(1180,150): alarm colour if CARGADO2; x offset x2; y offset y2
ellipse at (1110,140)-(1131,161): x offset x2; y offset y2
ellipse at (1150,140)-(1171,161): x offset x2; y offset y2
ellipse at (480,540)-(521,581): alarm colour if .SEM_SAL_REAL
ellipse at (480,380)-(521,421): alarm colour if .LLENO OR .SEM_ENT_COC
27 more shapes without text or variables
11 elements of other kinds (tables, trends, ...) not read
*)
